(* Visualisation VISU_CFG_KEEL
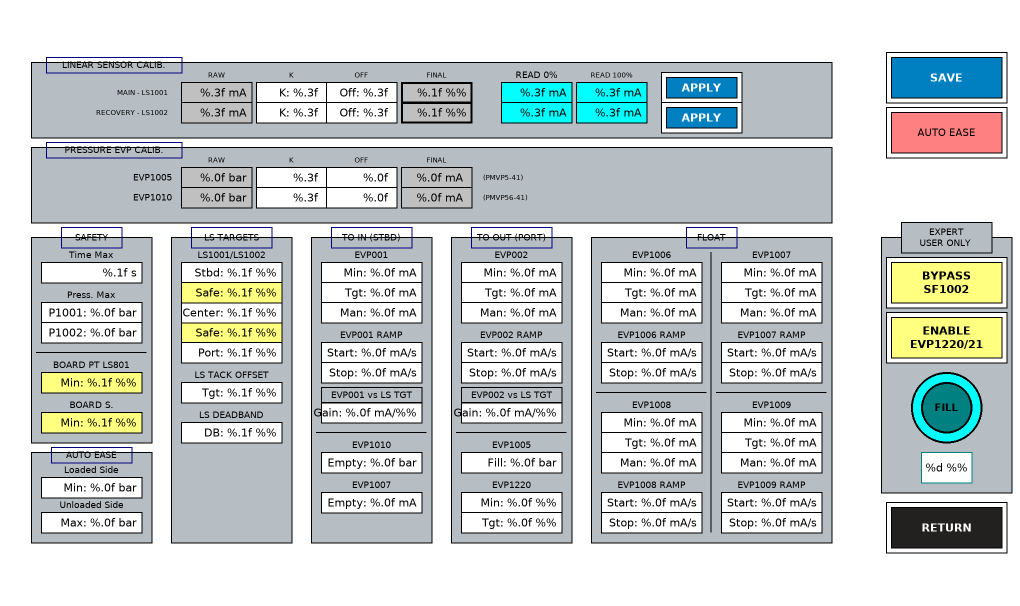
rectangle at (415,65)-(486,81): text "FINAL"
rectangle at (485,225)-(566,246): text "TO OUT (PORT)"
rectangle at (345,225)-(426,246): text "TO IN (STBD)"
rectangle at (20,550)-(331,601): text "%s"; shows INPUTS.sVisuTime
rounded rectangle at (905,55)-(1016,96): text "SAVE"; alarm colour if PARAMS.Save; toggles PARAMS.Save
rounded rectangle at (905,505)-(1016,546): text "RETURN"; opens VISU_2_KEEL
rectangle at (730,550)-(896,601): text "SAVED!"; invisible if PARAMS.Saved
rectangle at (20,0)-(426,51): text "CFG: KEEL"
rectangle at (55,260)-(156,281): text "%.1f s"; shows PARAMS.stKeelCfg.TimeMax; runs INTERN ASSIGN INPUTS.PresSelCalStbd[9]:=(FALSE); editable
rectangle at (65,245)-(146,261): text "Time Max"
rectangle at (55,300)-(156,321): text "P1001: %.0f bar"; shows P1001.MaxBar; runs INTERN ASSIGN INPUTS.PresSelCalStbd[9]:=(FALSE); editable
rectangle at (55,285)-(156,301): text "Press. Max"
rectangle at (55,320)-(156,341): text "P1002: %.0f bar"; shows P1002.MaxBar; runs INTERN ASSIGN INPUTS.PresSelCalStbd[9]:=(FALSE); editable
rectangle at (195,150)-(266,166): text "RAW"
rectangle at (415,150)-(486,166): text "FINAL"
rectangle at (270,150)-(341,166): text "K"
rectangle at (340,150)-(411,166): text "OFF"
rectangle at (415,165)-(486,186): text "%.0f mA"; shows EVP1005.mA; runs INTERN ASSIGN INPUTS.PresSelCalStbd[9]:=(FALSE)
rectangle at (270,165)-(341,186): text "%.3f"; shows EVP1005.Cal_K; runs INTERN ASSIGN INPUTS.PresSelCalStbd[9]:=(FALSE); editable
rectangle at (195,165)-(266,186): text "%.0f bar"; shows EVP1005.Bar; runs INTERN ASSIGN INPUTS.PresSelCalStbd[9]:=(FALSE)
rectangle at (340,165)-(411,186): text "%.0f"; shows EVP1005.Cal_Off; runs INTERN ASSIGN INPUTS.PresSelCalStbd[9]:=(FALSE); editable
rectangle at (145,165)-(196,186): text "EVP1005"
rectangle at (415,185)-(486,206): text "%.0f mA"; shows EVP1010.mA; runs INTERN ASSIGN INPUTS.PresSelCalStbd[9]:=(FALSE)
rectangle at (270,185)-(341,206): text "%.3f"; shows EVP1010.Cal_K; runs INTERN ASSIGN INPUTS.PresSelCalStbd[9]:=(FALSE); editable
rectangle at (195,185)-(266,206): text "%.0f bar"; shows EVP1010.Bar; runs INTERN ASSIGN INPUTS.PresSelCalStbd[9]:=(FALSE)
rectangle at (340,185)-(411,206): text "%.0f"; shows EVP1010.Cal_Off; runs INTERN ASSIGN INPUTS.PresSelCalStbd[9]:=(FALSE); editable
rectangle at (495,165)-(561,186): text "(PMVP5-41)"
rectangle at (145,185)-(196,206): text "EVP1010"
rectangle at (495,185)-(561,206): text "(PMVP56-41)"
ellipse at (925,370)-(996,441): alarm colour if MAIN.fbKeel.EVP_Fill = 0
ellipse at (935,380)-(986,431): text "FILL"; alarm colour if MAIN.fbKeel.IN_Hmi_fill; taps MAIN.fbKeel.IN_Hmi_fill
rounded rectangle at (905,315)-(1016,356): text "ENABLE / EVP1220/21"; alarm colour if MAIN.fbKEEL.EnableFill; toggles MAIN.fbKEEL.EnableFill
rounded rectangle at (915,220)-(1006,251): text "EXPERT / USER ONLY"
rounded rectangle at (680,75)-(751,96): text "APPLY"; toggles LS1001.Cal_Apply
rectangle at (590,80)-(661,101): text "%.3f mA"; shows LS1001.Cal_Max; alarm colour if LS1001.Cal_Max = 0.0; runs INTERN ASSIGN INPUTS.PresSelCalStbd[9]:=(FALSE); editable
rectangle at (515,80)-(586,101): text "%.3f mA"; shows LS1001.Cal_Min; alarm colour if LS1001.Cal_Min = 0.0; runs INTERN ASSIGN INPUTS.PresSelCalStbd[9]:=(FALSE); editable
rectangle at (55,80)-(186,101): text "MAIN - LS1001"
rectangle at (270,80)-(341,101): text "K: %.3f"; shows LS1001.Cal_K; runs INTERN ASSIGN INPUTS.PresSelCalStbd[9]:=(FALSE); editable
rectangle at (195,80)-(266,101): text "%.3f mA"; shows LS1001.Raw; alarm colour if LS1001.Err; runs INTERN ASSIGN INPUTS.PresSelCalStbd[9]:=(FALSE)
rectangle at (340,80)-(411,101): text "Off: %.3f"; shows LS1001.Cal_Off; runs INTERN ASSIGN INPUTS.PresSelCalStbd[9]:=(FALSE); editable
rectangle at (415,80)-(486,101): text "%.1f %%"; shows LS1001.Pos; runs INTERN ASSIGN INPUTS.PresSelCalStbd[9]:=(FALSE)
rectangle at (515,65)-(586,81): text "READ 0%"
rectangle at (590,65)-(661,81): text "READ 100%"
rounded rectangle at (680,105)-(751,126): text "APPLY"; toggles LS1002.Cal_Apply
rectangle at (590,100)-(661,121): text "%.3f mA"; shows LS1002.Cal_Max; alarm colour if LS1002.Cal_Max = 0.0; runs INTERN ASSIGN INPUTS.PresSelCalStbd[9]:=(FALSE); editable
rectangle at (515,100)-(586,121): text "%.3f mA"; shows LS1002.Cal_Min; alarm colour if LS1002.Cal_Min = 0.0; runs INTERN ASSIGN INPUTS.PresSelCalStbd[9]:=(FALSE); editable
rectangle at (55,100)-(186,121): text "RECOVERY - LS1002"
rectangle at (270,100)-(341,121): text "K: %.3f"; shows LS1002.Cal_K; runs INTERN ASSIGN INPUTS.PresSelCalStbd[9]:=(FALSE); editable
rectangle at (195,100)-(266,121): text "%.3f mA"; shows LS1002.Raw; alarm colour if LS1002.Err; runs INTERN ASSIGN INPUTS.PresSelCalStbd[9]:=(FALSE)
rectangle at (340,100)-(411,121): text "Off: %.3f"; shows LS1002.Cal_Off; runs INTERN ASSIGN INPUTS.PresSelCalStbd[9]:=(FALSE); editable
rectangle at (415,100)-(486,121): text "%.1f %%"; shows LS1002.Pos; runs INTERN ASSIGN INPUTS.PresSelCalStbd[9]:=(FALSE)
rounded rectangle at (905,260)-(1016,301): text "BYPASS / SF1002"; alarm colour if MAIN.fbKEEL.BypassSF; toggles MAIN.fbKEEL.BypassSF
rectangle at (55,370)-(156,391): text "Min: %.1f %%"; shows PARAMS.stKeelCfg.Board_P_Min_Out; runs INTERN ASSIGN INPUTS.PresSelCalStbd[9]:=(FALSE); editable
rectangle at (55,355)-(156,371): text "BOARD PT LS801"
rectangle at (55,410)-(156,431): text "Min: %.1f %%"; shows PARAMS.stKeelCfg.Board_S_Min_Out; runs INTERN ASSIGN INPUTS.PresSelCalStbd[9]:=(FALSE); editable
rectangle at (55,395)-(156,411): text "BOARD S."
rounded rectangle at (935,450)-(986,481): text "%d %%"; shows MAIN.fbKEEL.IN_Hmi_fill_Perc; editable 5..100
rectangle at (195,260)-(296,281): text "Stbd: %.1f %%"; shows PARAMS.stKeelCfg.TgtLS_In; runs INTERN ASSIGN INPUTS.PresSelCalStbd[9]:=(FALSE); editable
rectangle at (195,245)-(296,261): text "LS1001/LS1002"
rectangle at (195,320)-(296,341): text "Safe: %.1f %%"; shows PARAMS.stKeelCfg.TgtLS_Safe_Out; runs INTERN ASSIGN INPUTS.PresSelCalStbd[9]:=(FALSE); editable
rectangle at (195,300)-(296,321): text "Center: %.1f %%"; shows PARAMS.stKeelCfg.TgtLS_Mid; runs INTERN ASSIGN INPUTS.PresSelCalStbd[9]:=(FALSE); editable
rectangle at (195,280)-(296,301): text "Safe: %.1f %%"; shows PARAMS.stKeelCfg.TgtLS_Safe_In; runs INTERN ASSIGN INPUTS.PresSelCalStbd[9]:=(FALSE); editable
rectangle at (195,340)-(296,361): text "Port: %.1f %%"; shows PARAMS.stKeelCfg.TgtLS_Out; runs INTERN ASSIGN INPUTS.PresSelCalStbd[9]:=(FALSE); editable
rectangle at (195,420)-(296,441): text "DB: %.1f %%"; shows PARAMS.stKeelCfg.LS_DB; runs INTERN ASSIGN INPUTS.PresSelCalStbd[9]:=(FALSE); editable
rectangle at (195,405)-(296,421): text "LS DEADBAND"
rectangle at (615,260)-(716,281): text "Min: %.0f mA"; shows PARAMS.stKeelCfg.EVP_In_SE_Min; runs INTERN ASSIGN INPUTS.PresSelCalStbd[9]:=(FALSE); editable
rectangle at (615,245)-(716,261): text "EVP1006"
rectangle at (615,280)-(716,301): text "Tgt: %.0f mA"; shows PARAMS.stKeelCfg.EVP_In_SE_Max; runs INTERN ASSIGN INPUTS.PresSelCalStbd[9]:=(FALSE); editable
rectangle at (615,300)-(716,321): text "Man: %.0f mA"; shows PARAMS.stKeelCfg.EVP_In_SE_Man; runs INTERN ASSIGN INPUTS.PresSelCalStbd[9]:=(FALSE); editable
rectangle at (615,410)-(716,431): text "Min: %.0f mA"; shows PARAMS.stKeelCfg.EVP_In_FE_Min; runs INTERN ASSIGN INPUTS.PresSelCalStbd[9]:=(FALSE); editable
rectangle at (615,395)-(716,411): text "EVP1008"
rectangle at (615,430)-(716,451): text "Tgt: %.0f mA"; shows PARAMS.stKeelCfg.EVP_In_FE_Max; runs INTERN ASSIGN INPUTS.PresSelCalStbd[9]:=(FALSE); editable
rectangle at (615,450)-(716,471): text "Man: %.0f mA"; shows PARAMS.stKeelCfg.EVP_In_FE_Man; runs INTERN ASSIGN INPUTS.PresSelCalStbd[9]:=(FALSE); editable
rectangle at (335,260)-(436,281): text "Min: %.0f mA"; shows PARAMS.stKeelCfg.EVP_In_Eng_Min; runs INTERN ASSIGN INPUTS.PresSelCalStbd[9]:=(FALSE); editable
rectangle at (335,245)-(436,261): text "EVP001"
rectangle at (335,280)-(436,301): text "Tgt: %.0f mA"; shows PARAMS.stKeelCfg.EVP_In_Eng_Max; runs INTERN ASSIGN INPUTS.PresSelCalStbd[9]:=(FALSE); editable
rectangle at (335,300)-(436,321): text "Man: %.0f mA"; shows PARAMS.stKeelCfg.EVP_In_Eng_Man; runs INTERN ASSIGN INPUTS.PresSelCalStbd[9]:=(FALSE); editable
rectangle at (335,490)-(436,511): text "Empty: %.0f mA"; shows PARAMS.stKeelCfg.EVP_Out_SE_Empty; runs INTERN ASSIGN INPUTS.PresSelCalStbd[9]:=(FALSE); editable
rectangle at (335,475)-(436,491): text "EVP1007"
rectangle at (195,380)-(296,401): text "Tgt: %.1f %%"; shows PARAMS.stKeelCfg.TgtLS_Tack_Off; runs INTERN ASSIGN INPUTS.PresSelCalStbd[9]:=(FALSE); editable
rectangle at (195,365)-(296,381): text "LS TACK OFFSET"
rectangle at (335,450)-(436,471): text "Empty: %.0f bar"; shows PARAMS.stKeelCfg.EVP_In_P_Empty; runs INTERN ASSIGN INPUTS.PresSelCalStbd[9]:=(FALSE); editable
rectangle at (335,435)-(436,451): text "EVP1010"
rectangle at (475,260)-(576,281): text "Min: %.0f mA"; shows PARAMS.stKeelCfg.EVP_Out_Eng_Min; runs INTERN ASSIGN INPUTS.PresSelCalStbd[9]:=(FALSE); editable
rectangle at (475,245)-(576,261): text "EVP002"
rectangle at (475,280)-(576,301): text "Tgt: %.0f mA"; shows PARAMS.stKeelCfg.EVP_Out_Eng_Max; runs INTERN ASSIGN INPUTS.PresSelCalStbd[9]:=(FALSE); editable
rectangle at (475,300)-(576,321): text "Man: %.0f mA"; shows PARAMS.stKeelCfg.EVP_Out_Eng_Man; runs INTERN ASSIGN INPUTS.PresSelCalStbd[9]:=(FALSE); editable
rectangle at (475,450)-(576,471): text "Fill: %.0f bar"; shows PARAMS.stKeelCfg.EVP_Out_P_Fill; runs INTERN ASSIGN INPUTS.PresSelCalStbd[9]:=(FALSE); editable
rectangle at (475,435)-(576,451): text "EVP1005"
rectangle at (475,490)-(576,511): text "Min: %.0f %%"; shows PARAMS.stKeelCfg.EVP_Out_Fill_Min; runs INTERN ASSIGN INPUTS.PresSelCalStbd[9]:=(FALSE); editable
rectangle at (475,475)-(576,491): text "EVP1220"
rectangle at (475,510)-(576,531): text "Tgt: %.0f %%"; shows PARAMS.stKeelCfg.EVP_Out_Fill_Max; runs INTERN ASSIGN INPUTS.PresSelCalStbd[9]:=(FALSE); editable
rectangle at (735,260)-(836,281): text "Min: %.0f mA"; shows PARAMS.stKeelCfg.EVP_Out_SE_Min; runs INTERN ASSIGN INPUTS.PresSelCalStbd[9]:=(FALSE); editable
rectangle at (735,245)-(836,261): text "EVP1007"
rectangle at (735,280)-(836,301): text "Tgt: %.0f mA"; shows PARAMS.stKeelCfg.EVP_Out_SE_Max; runs INTERN ASSIGN INPUTS.PresSelCalStbd[9]:=(FALSE); editable
rectangle at (735,300)-(836,321): text "Man: %.0f mA"; shows PARAMS.stKeelCfg.EVP_Out_SE_Man; runs INTERN ASSIGN INPUTS.PresSelCalStbd[9]:=(FALSE); editable
rectangle at (735,410)-(836,431): text "Min: %.0f mA"; shows PARAMS.stKeelCfg.EVP_Out_FE_Min; runs INTERN ASSIGN INPUTS.PresSelCalStbd[9]:=(FALSE); editable
rectangle at (735,395)-(836,411): text "EVP1009"
rectangle at (735,430)-(836,451): text "Tgt: %.0f mA"; shows PARAMS.stKeelCfg.EVP_Out_FE_Max; runs INTERN ASSIGN INPUTS.PresSelCalStbd[9]:=(FALSE); editable
rectangle at (735,450)-(836,471): text "Man: %.0f mA"; shows PARAMS.stKeelCfg.EVP_Out_FE_Man; runs INTERN ASSIGN INPUTS.PresSelCalStbd[9]:=(FALSE); editable
rectangle at (335,340)-(436,361): text "Start: %.0f mA/s"; shows PARAMS.stKeelCfg.EVP_In_Eng_Inc; runs INTERN ASSIGN INPUTS.PresSelCalStbd[9]:=(FALSE); editable
rectangle at (335,325)-(436,341): text "EVP001 RAMP"
rectangle at (335,360)-(436,381): text "Stop: %.0f mA/s"; shows PARAMS.stKeelCfg.EVP_In_Eng_Dec; runs INTERN ASSIGN INPUTS.PresSelCalStbd[9]:=(FALSE); editable
rectangle at (475,340)-(576,361): text "Start: %.0f mA/s"; shows PARAMS.stKeelCfg.EVP_Out_Eng_Inc; runs INTERN ASSIGN INPUTS.PresSelCalStbd[9]:=(FALSE); editable
rectangle at (475,325)-(576,341): text "EVP002 RAMP"
rectangle at (475,360)-(576,381): text "Stop: %.0f mA/s"; shows PARAMS.stKeelCfg.EVP_Out_Eng_Dec; runs INTERN ASSIGN INPUTS.PresSelCalStbd[9]:=(FALSE); editable
rectangle at (615,340)-(716,361): text "Start: %.0f mA/s"; shows PARAMS.stKeelCfg.EVP_In_SE_Inc; runs INTERN ASSIGN INPUTS.PresSelCalStbd[9]:=(FALSE); editable
rectangle at (615,325)-(716,341): text "EVP1006 RAMP"
rectangle at (615,360)-(716,381): text "Stop: %.0f mA/s"; shows PARAMS.stKeelCfg.EVP_In_SE_Dec; runs INTERN ASSIGN INPUTS.PresSelCalStbd[9]:=(FALSE); editable
rectangle at (735,340)-(836,361): text "Start: %.0f mA/s"; shows PARAMS.stKeelCfg.EVP_Out_SE_Inc; runs INTERN ASSIGN INPUTS.PresSelCalStbd[9]:=(FALSE); editable
rectangle at (735,325)-(836,341): text "EVP1007 RAMP"
rectangle at (735,360)-(836,381): text "Stop: %.0f mA/s"; shows PARAMS.stKeelCfg.EVP_Out_SE_Dec; runs INTERN ASSIGN INPUTS.PresSelCalStbd[9]:=(FALSE); editable
rectangle at (615,490)-(716,511): text "Start: %.0f mA/s"; shows PARAMS.stKeelCfg.EVP_In_FE_Inc; runs INTERN ASSIGN INPUTS.PresSelCalStbd[9]:=(FALSE); editable
rectangle at (615,475)-(716,491): text "EVP1008 RAMP"
rectangle at (615,510)-(716,531): text "Stop: %.0f mA/s"; shows PARAMS.stKeelCfg.EVP_In_FE_Dec; runs INTERN ASSIGN INPUTS.PresSelCalStbd[9]:=(FALSE); editable
rectangle at (735,490)-(836,511): text "Start: %.0f mA/s"; shows PARAMS.stKeelCfg.EVP_Out_FE_Inc; runs INTERN ASSIGN INPUTS.PresSelCalStbd[9]:=(FALSE); editable
rectangle at (735,475)-(836,491): text "EVP1009 RAMP"
rectangle at (735,510)-(836,531): text "Stop: %.0f mA/s"; shows PARAMS.stKeelCfg.EVP_Out_FE_Dec; runs INTERN ASSIGN INPUTS.PresSelCalStbd[9]:=(FALSE); editable
rectangle at (335,400)-(436,421): text "Gain: %.0f mA/%%"; shows PARAMS.stKeelCfg.EVP_In_Eng_K; runs INTERN ASSIGN INPUTS.PresSelCalStbd[9]:=(FALSE); editable
rectangle at (335,385)-(436,401): text "EVP001 vs LS TGT"
rectangle at (475,400)-(576,421): text "Gain: %.0f mA/%%"; shows PARAMS.stKeelCfg.EVP_Out_Eng_K; runs INTERN ASSIGN INPUTS.PresSelCalStbd[9]:=(FALSE); editable
rectangle at (475,385)-(576,401): text "EVP002 vs LS TGT"
rectangle at (700,225)-(751,246): text "FLOAT"
rectangle at (195,65)-(266,81): text "RAW"
rectangle at (270,65)-(341,81): text "K"
rectangle at (340,65)-(411,81): text "OFF"
rectangle at (205,225)-(286,246): text "LS TARGETS"
rectangle at (75,225)-(136,246): text "SAFETY"
rectangle at (60,55)-(196,71): text "LINEAR SENSOR CALIB."
rectangle at (60,140)-(196,156): text "PRESSURE EVP CALIB."
rounded rectangle at (905,110)-(1016,151): text "AUTO EASE"; alarm colour if MAIN.aLP_Enable[20]; toggles MAIN.aLP_Enable[20]
rectangle at (65,445)-(146,461): text "AUTO EASE"
rectangle at (55,460)-(156,476): text "Loaded Side"
rectangle at (55,475)-(156,496): text "Min: %.0f bar"; shows PARAMS.stKeelCfg.MinLoadSide_Bar; runs INTERN ASSIGN INPUTS.PresSelCalStbd[9]:=(FALSE); editable
rectangle at (55,495)-(156,511): text "Unloaded Side"
rectangle at (55,510)-(156,531): text "Max: %.0f bar"; shows PARAMS.stKeelCfg.MaxUnloadSide_Bar; runs INTERN ASSIGN INPUTS.PresSelCalStbd[9]:=(FALSE); editable
22 more shapes without text or variables
*)

(* Visualisation VISU_CFG_POWERPACK
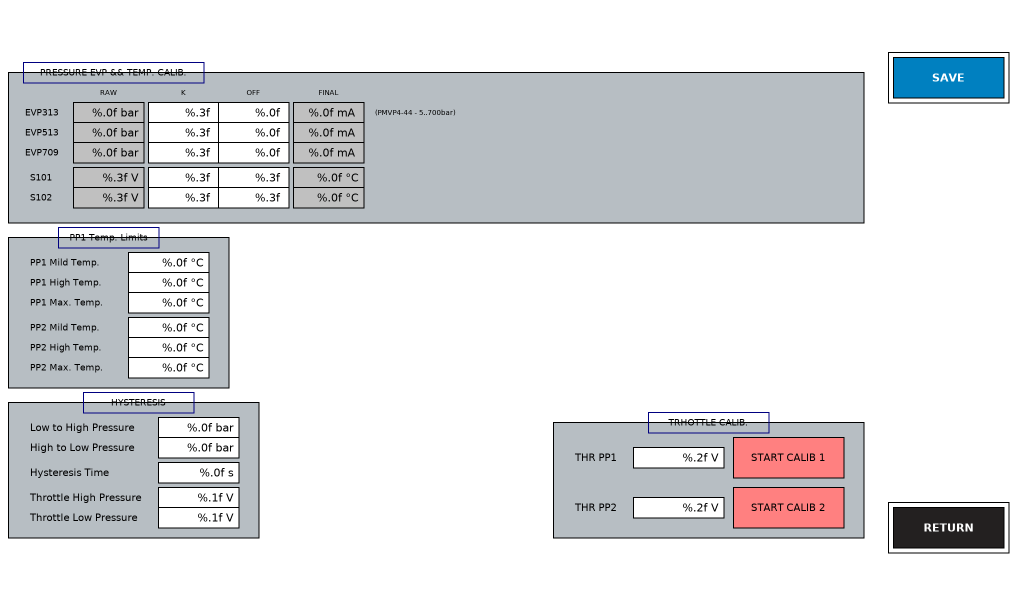
rectangle at (20,0)-(436,51): text "CFG: POWERPACK"
rectangle at (20,550)-(331,601): text "%s"; shows INPUTS.sVisuTime
rounded rectangle at (905,55)-(1016,96): text "SAVE"; alarm colour if PARAMS.Save; toggles PARAMS.Save
rounded rectangle at (905,505)-(1016,546): text "RETURN"; opens VISU_1_PUMPS
rectangle at (95,390)-(206,411): text "HYSTERESIS"
rectangle at (170,415)-(251,436): text "%.0f bar"; shows PARAMS.stPowerpackCfg.Hyst_HP; runs INTERN ASSIGN INPUTS.PresSelCalStbd[9]:=(FALSE); editable
rectangle at (170,435)-(251,456): text "%.0f bar"; shows PARAMS.stPowerpackCfg.Hyst_LP; runs INTERN ASSIGN INPUTS.PresSelCalStbd[9]:=(FALSE); editable
rectangle at (170,460)-(251,481): text "%.0f s"; shows PARAMS.stPowerpackCfg.Hyst_TM; runs INTERN ASSIGN INPUTS.PresSelCalStbd[9]:=(FALSE); editable
rectangle at (40,415)-(171,436): text "Low to High Pressure"; shows RECV_J1939.F004.DriverDemandTorque
rectangle at (40,435)-(171,456): text "High to Low Pressure"; shows RECV_J1939.F004.DriverDemandTorque
rectangle at (40,460)-(171,481): text "Hysteresis Time"; shows RECV_J1939.F004.DriverDemandTorque
rectangle at (730,550)-(896,601): text "SAVED!"; invisible if PARAMS.Saved
rectangle at (660,410)-(781,431): text "TRHOTTLE CALIB."
rounded rectangle at (745,435)-(856,476): text "START CALIB 1"; alarm colour if POWERPACK.Calib1; toggles POWERPACK.Calib1
rectangle at (645,445)-(736,466): text "%.2f V"; shows THR_PP1; runs INTERN ASSIGN INPUTS.PresSelCalStbd[9]:=(FALSE); editable
rectangle at (585,445)-(641,466): text "THR PP1"; shows RECV_J1939.F004.DriverDemandTorque
rectangle at (645,495)-(736,516): text "%.2f V"; shows THR_PP2; runs INTERN ASSIGN INPUTS.PresSelCalStbd[9]:=(FALSE); editable
rectangle at (585,495)-(641,516): text "THR PP2"; shows RECV_J1939.F004.DriverDemandTorque
rounded rectangle at (745,485)-(856,526): text "START CALIB 2"; alarm colour if POWERPACK.Calib2; toggles POWERPACK.Calib2
rectangle at (170,485)-(251,506): text "%.1f V"; shows PARAMS.stPowerpackCfg.Thr_HP; runs INTERN ASSIGN INPUTS.PresSelCalStbd[9]:=(FALSE); editable 1..5
rectangle at (40,485)-(171,506): text "Throttle High Pressure"; shows RECV_J1939.F004.DriverDemandTorque
rectangle at (170,505)-(251,526): text "%.1f V"; shows PARAMS.stPowerpackCfg.Thr_LP; runs INTERN ASSIGN INPUTS.PresSelCalStbd[9]:=(FALSE); editable 1..5
rectangle at (40,505)-(171,526): text "Throttle Low Pressure"; shows RECV_J1939.F004.DriverDemandTorque
rectangle at (85,80)-(156,101): text "RAW"
rectangle at (305,80)-(376,101): text "FINAL"
rectangle at (160,80)-(231,101): text "K"
rectangle at (230,80)-(301,101): text "OFF"
rectangle at (305,100)-(376,121): text "%.0f mA"; shows EVP313.mA; runs INTERN ASSIGN INPUTS.PresSelCalStbd[9]:=(FALSE)
rectangle at (160,100)-(231,121): text "%.3f"; shows EVP313.Cal_K; runs INTERN ASSIGN INPUTS.PresSelCalStbd[9]:=(FALSE); editable
rectangle at (85,100)-(156,121): text "%.0f bar"; shows EVP313.Bar; runs INTERN ASSIGN INPUTS.PresSelCalStbd[9]:=(FALSE)
rectangle at (230,100)-(301,121): text "%.0f"; shows EVP313.Cal_Off; runs INTERN ASSIGN INPUTS.PresSelCalStbd[9]:=(FALSE); editable
rectangle at (35,100)-(86,121): text "EVP313"
rectangle at (305,120)-(376,141): text "%.0f mA"; shows EVP513.mA; runs INTERN ASSIGN INPUTS.PresSelCalStbd[9]:=(FALSE)
rectangle at (160,120)-(231,141): text "%.3f"; shows EVP513.Cal_K; runs INTERN ASSIGN INPUTS.PresSelCalStbd[9]:=(FALSE); editable
rectangle at (85,120)-(156,141): text "%.0f bar"; shows EVP513.Bar; runs INTERN ASSIGN INPUTS.PresSelCalStbd[9]:=(FALSE)
rectangle at (230,120)-(301,141): text "%.0f"; shows EVP513.Cal_Off; runs INTERN ASSIGN INPUTS.PresSelCalStbd[9]:=(FALSE); editable
rectangle at (385,100)-(581,121): text "(PMVP4-44 - 5..700bar)"
rectangle at (305,140)-(376,161): text "%.0f mA"; shows EVP709.mA; runs INTERN ASSIGN INPUTS.PresSelCalStbd[9]:=(FALSE)
rectangle at (160,140)-(231,161): text "%.3f"; shows EVP709.Cal_K; runs INTERN ASSIGN INPUTS.PresSelCalStbd[9]:=(FALSE); editable
rectangle at (85,140)-(156,161): text "%.0f bar"; shows EVP709.Bar; runs INTERN ASSIGN INPUTS.PresSelCalStbd[9]:=(FALSE)
rectangle at (230,140)-(301,161): text "%.0f"; shows EVP709.Cal_Off; runs INTERN ASSIGN INPUTS.PresSelCalStbd[9]:=(FALSE); editable
rectangle at (35,120)-(86,141): text "EVP513"
rectangle at (35,140)-(86,161): text "EVP709"
rectangle at (35,60)-(216,81): text "PRESSURE EVP && TEMP. CALIB."
rectangle at (40,250)-(121,271): text "PP1 Mild Temp."
rectangle at (140,250)-(221,271): text "%.0f °C"; shows S101.LowDeg; runs INTERN ASSIGN INPUTS.PresSelCalStbd[9]:=(FALSE); editable
rectangle at (40,270)-(121,291): text "PP1 High Temp."
rectangle at (140,270)-(221,291): text "%.0f °C"; shows S101.HigDeg; runs INTERN ASSIGN INPUTS.PresSelCalStbd[9]:=(FALSE); editable
rectangle at (70,225)-(171,246): text "PP1 Temp. Limits"
rectangle at (40,290)-(121,311): text "PP1 Max. Temp."
rectangle at (140,290)-(221,311): text "%.0f °C"; shows S101.MaxDeg; runs INTERN ASSIGN INPUTS.PresSelCalStbd[9]:=(FALSE); editable
rectangle at (40,165)-(86,186): text "S101"
rectangle at (305,165)-(376,186): text "%.0f °C"; shows S101.Deg
rectangle at (160,165)-(231,186): text "%.3f"; shows S101.Cal_K; runs INTERN ASSIGN INPUTS.PresSelCalStbd[9]:=(FALSE); editable
rectangle at (85,165)-(156,186): text "%.3f V"; shows S101.Raw; alarm colour if S101.Err; runs INTERN ASSIGN INPUTS.PresSelCalStbd[9]:=(FALSE)
rectangle at (230,165)-(301,186): text "%.3f"; shows S101.Cal_Off; runs INTERN ASSIGN INPUTS.PresSelCalStbd[9]:=(FALSE); editable
rectangle at (40,185)-(86,206): text "S102"
rectangle at (305,185)-(376,206): text "%.0f °C"; shows S102.Deg
rectangle at (160,185)-(231,206): text "%.3f"; shows S102.Cal_K; runs INTERN ASSIGN INPUTS.PresSelCalStbd[9]:=(FALSE); editable
rectangle at (85,185)-(156,206): text "%.3f V"; shows S102.Raw; alarm colour if S102.Err; runs INTERN ASSIGN INPUTS.PresSelCalStbd[9]:=(FALSE)
rectangle at (230,185)-(301,206): text "%.3f"; shows S102.Cal_Off; runs INTERN ASSIGN INPUTS.PresSelCalStbd[9]:=(FALSE); editable
rectangle at (40,315)-(121,336): text "PP2 Mild Temp."
rectangle at (140,315)-(221,336): text "%.0f °C"; shows S102.LowDeg; runs INTERN ASSIGN INPUTS.PresSelCalStbd[9]:=(FALSE); editable
rectangle at (40,335)-(121,356): text "PP2 High Temp."
rectangle at (140,335)-(221,356): text "%.0f °C"; shows S102.HigDeg; runs INTERN ASSIGN INPUTS.PresSelCalStbd[9]:=(FALSE); editable
rectangle at (40,355)-(121,376): text "PP2 Max. Temp."
rectangle at (140,355)-(221,376): text "%.0f °C"; shows S102.MaxDeg; runs INTERN ASSIGN INPUTS.PresSelCalStbd[9]:=(FALSE); editable
6 more shapes without text or variables
*)

(* Visualisation VISU_CFG_PROPULSION
rectangle at (55,305)-(116,326): text "PROP"
rounded rectangle at (905,505)-(1016,546): text "RETURN"; opens VISU_1_ENGINE
rectangle at (20,0)-(331,51): text "CFG: PROPULSION"
rectangle at (305,185)-(376,206): text "%.0f rpm"; shows PARAMS.stPropulsionCfg.aEng_RPM[10]; editable
rectangle at (380,185)-(451,206): text "%.0f mA"; shows PARAMS.stPropulsionCfg.aEVP_mA[10]; editable
rectangle at (195,185)-(226,206): text "100%"
rectangle at (230,185)-(301,206): text "%.2f V"; shows PARAMS.stPropulsionCfg.aThrt_V[10]; runs INTERN ASSIGN INPUTS.PresSelCalStbd[9]:=(FALSE); editable
rectangle at (230,365)-(301,386): text "%.2f V"; shows PARAMS.stPropulsionCfg.aThrt_V[0]; runs INTERN ASSIGN INPUTS.PresSelCalStbd[9]:=(FALSE); editable
rectangle at (195,105)-(226,126): text "0%"
rectangle at (230,105)-(301,126): text "%.2f V"; shows PARAMS.stPropulsionCfg.aThrt_V[6]; editable
rectangle at (230,285)-(301,306): text "%.2f V"; shows PARAMS.stPropulsionCfg.aThrt_V[4]; runs INTERN ASSIGN INPUTS.PresSelCalStbd[9]:=(FALSE); editable
rectangle at (195,165)-(226,186): text "75%"
rectangle at (195,145)-(226,166): text "50%"
rectangle at (195,125)-(226,146): text "25%"
rectangle at (230,85)-(301,106): text "THROTTLE"
rectangle at (305,85)-(376,106): text "ENGINE"
rectangle at (380,85)-(451,106): text "PROPELLER"
rectangle at (305,165)-(376,186): text "%.0f rpm"; shows PARAMS.stPropulsionCfg.aEng_RPM[9]; editable
rectangle at (305,145)-(376,166): text "%.0f rpm"; shows PARAMS.stPropulsionCfg.aEng_RPM[8]; editable
rectangle at (305,125)-(376,146): text "%.0f rpm"; shows PARAMS.stPropulsionCfg.aEng_RPM[7]; editable
rectangle at (305,105)-(376,126): text "%.0f rpm"; shows PARAMS.stPropulsionCfg.aEng_RPM[6]; editable
rectangle at (305,285)-(376,306): text "%.0f rpm"; shows PARAMS.stPropulsionCfg.aEng_RPM[4]; editable
rectangle at (305,305)-(376,326): text "%.0f rpm"; shows PARAMS.stPropulsionCfg.aEng_RPM[3]; editable
rectangle at (305,325)-(376,346): text "%.0f rpm"; shows PARAMS.stPropulsionCfg.aEng_RPM[2]; editable
rectangle at (305,345)-(376,366): text "%.0f rpm"; shows PARAMS.stPropulsionCfg.aEng_RPM[1]; editable
rectangle at (305,365)-(376,386): text "%.0f rpm"; shows PARAMS.stPropulsionCfg.aEng_RPM[0]; editable
rectangle at (230,125)-(301,146): text "%.2f V"; shows PARAMS.stPropulsionCfg.aThrt_V[7]
rectangle at (230,145)-(301,166): text "%.2f V"; shows PARAMS.stPropulsionCfg.aThrt_V[8]
rectangle at (230,165)-(301,186): text "%.2f V"; shows PARAMS.stPropulsionCfg.aThrt_V[9]
rectangle at (230,305)-(301,326): text "%.2f V"; shows PARAMS.stPropulsionCfg.aThrt_V[3]
rectangle at (230,325)-(301,346): text "%.2f V"; shows PARAMS.stPropulsionCfg.aThrt_V[2]
rectangle at (230,345)-(301,366): text "%.2f V"; shows PARAMS.stPropulsionCfg.aThrt_V[1]
rectangle at (380,165)-(451,186): text "%.0f mA"; shows PARAMS.stPropulsionCfg.aEVP_mA[9]; editable
rectangle at (380,145)-(451,166): text "%.0f mA"; shows PARAMS.stPropulsionCfg.aEVP_mA[8]; editable
rectangle at (380,125)-(451,146): text "%.0f mA"; shows PARAMS.stPropulsionCfg.aEVP_mA[7]; editable
rectangle at (380,105)-(451,126): text "%.0f mA"; shows PARAMS.stPropulsionCfg.aEVP_mA[6]; editable
rectangle at (380,285)-(451,306): text "%.0f mA"; shows PARAMS.stPropulsionCfg.aEVP_mA[4]; editable
rectangle at (290,240)-(391,261): text "REVERSE"
rectangle at (380,305)-(451,326): text "%.0f mA"; shows PARAMS.stPropulsionCfg.aEVP_mA[3]; editable
rectangle at (380,325)-(451,346): text "%.0f mA"; shows PARAMS.stPropulsionCfg.aEVP_mA[2]; editable
rectangle at (380,345)-(451,366): text "%.0f mA"; shows PARAMS.stPropulsionCfg.aEVP_mA[1]; editable
rectangle at (380,365)-(451,386): text "%.0f mA"; shows PARAMS.stPropulsionCfg.aEVP_mA[0]; editable
rectangle at (0,0)-(1,1): text "{ExtendedElement},Visu\ElementDLL.ete,1,@Bargraph,76,131,1,1,0,PARAMS.stPropulsionCfg.aEng_RPM[10],,%,200,400,800,2400,0,0,0,0,0,0,0,-13,16,700,Arial,0,255,0,255,0,0,0,0,0,0,0,0,0,,0,"
rectangle at (12,65)-(28,122): alarm colour if (PARAMS.stPropulsionCfg.aEng_RPM[10]) < 0; top ((PARAMS.stPropulsionCfg.aEng_RPM[10] * 1.0) - 1600)  * -0.07125
rectangle at (0,0)-(1,1): text "{ExtendedElement},Visu\ElementDLL.ete,1,@Bargraph,76,131,1,1,0,PARAMS.stPropulsionCfg.aEng_RPM[9],,%,200,400,800,2400,0,0,0,0,0,0,0,-13,16,700,Arial,0,255,0,255,0,0,0,0,0,0,0,0,0,,0,"
rectangle at (12,65)-(28,122): alarm colour if (PARAMS.stPropulsionCfg.aEng_RPM[9]) < 0; top ((PARAMS.stPropulsionCfg.aEng_RPM[9] * 1.0) - 1600)  * -0.07125
rectangle at (0,0)-(1,1): text "{ExtendedElement},Visu\ElementDLL.ete,1,@Bargraph,76,131,1,1,0,PARAMS.stPropulsionCfg.aEng_RPM[8],,%,200,400,800,2400,0,0,0,0,0,0,0,-13,16,700,Arial,0,255,0,255,0,0,0,0,0,0,0,0,0,,0,"
rectangle at (12,65)-(28,122): alarm colour if (PARAMS.stPropulsionCfg.aEng_RPM[8]) < 0; top ((PARAMS.stPropulsionCfg.aEng_RPM[8] * 1.0) - 1600)  * -0.07125
rectangle at (0,0)-(1,1): text "{ExtendedElement},Visu\ElementDLL.ete,1,@Bargraph,76,131,1,1,0,PARAMS.stPropulsionCfg.aEng_RPM[7],,%,200,400,800,2400,0,0,0,0,0,0,0,-13,16,700,Arial,0,255,0,255,0,0,0,0,0,0,0,0,0,,0,"
rectangle at (12,65)-(28,122): alarm colour if (PARAMS.stPropulsionCfg.aEng_RPM[7]) < 0; top ((PARAMS.stPropulsionCfg.aEng_RPM[7] * 1.0) - 1600)  * -0.07125
rectangle at (0,0)-(1,1): text "{ExtendedElement},Visu\ElementDLL.ete,1,@Bargraph,76,131,1,1,0,PARAMS.stPropulsionCfg.aEng_RPM[6],,%,200,400,800,2400,0,0,0,0,0,0,0,-13,16,700,Arial,0,255,0,255,0,0,0,0,0,0,0,0,0,,0,"
rectangle at (12,65)-(28,122): alarm colour if (PARAMS.stPropulsionCfg.aEng_RPM[6]) < 0; top ((PARAMS.stPropulsionCfg.aEng_RPM[6] * 1.0) - 1600)  * -0.07125
rectangle at (455,80)-(486,101): text "2400"
rectangle at (455,110)-(486,131): text "2000"
rectangle at (455,140)-(486,161): text "1600"
rectangle at (455,170)-(486,191): text "1200"
rectangle at (455,200)-(486,221): text "800"
rectangle at (0,0)-(1,1): text "{ExtendedElement},Visu\ElementDLL.ete,1,@Bargraph,76,131,1,1,0,PARAMS.stPropulsionCfg.aEng_RPM[0],,%,200,400,800,2400,0,0,0,0,0,0,0,-13,16,700,Arial,0,255,0,255,0,0,0,0,0,0,0,0,0,,0,"
rectangle at (12,65)-(28,122): alarm colour if (PARAMS.stPropulsionCfg.aEng_RPM[0]) < 0; top ((PARAMS.stPropulsionCfg.aEng_RPM[0] * 1.0) - 1600)  * -0.07125
rectangle at (0,0)-(1,1): text "{ExtendedElement},Visu\ElementDLL.ete,1,@Bargraph,76,131,1,1,0,PARAMS.stPropulsionCfg.aEng_RPM[1],,%,200,400,800,2400,0,0,0,0,0,0,0,-13,16,700,Arial,0,255,0,255,0,0,0,0,0,0,0,0,0,,0,"
rectangle at (12,65)-(28,122): alarm colour if (PARAMS.stPropulsionCfg.aEng_RPM[1]) < 0; top ((PARAMS.stPropulsionCfg.aEng_RPM[1] * 1.0) - 1600)  * -0.07125
rectangle at (0,0)-(1,1): text "{ExtendedElement},Visu\ElementDLL.ete,1,@Bargraph,76,131,1,1,0,PARAMS.stPropulsionCfg.aEng_RPM[2],,%,200,400,800,2400,0,0,0,0,0,0,0,-13,16,700,Arial,0,255,0,255,0,0,0,0,0,0,0,0,0,,0,"
rectangle at (12,65)-(28,122): alarm colour if (PARAMS.stPropulsionCfg.aEng_RPM[2]) < 0; top ((PARAMS.stPropulsionCfg.aEng_RPM[2] * 1.0) - 1600)  * -0.07125
rectangle at (0,0)-(1,1): text "{ExtendedElement},Visu\ElementDLL.ete,1,@Bargraph,76,131,1,1,0,PARAMS.stPropulsionCfg.aEng_RPM[3],,%,200,400,800,2400,0,0,0,0,0,0,0,-13,16,700,Arial,0,255,0,255,0,0,0,0,0,0,0,0,0,,0,"
rectangle at (12,65)-(28,122): alarm colour if (PARAMS.stPropulsionCfg.aEng_RPM[3]) < 0; top ((PARAMS.stPropulsionCfg.aEng_RPM[3] * 1.0) - 1600)  * -0.07125
rectangle at (0,0)-(1,1): text "{ExtendedElement},Visu\ElementDLL.ete,1,@Bargraph,76,131,1,1,0,PARAMS.stPropulsionCfg.aEng_RPM[4],,%,200,400,800,2400,0,0,0,0,0,0,0,-13,16,700,Arial,0,255,0,255,0,0,0,0,0,0,0,0,0,,0,"
rectangle at (12,65)-(28,122): alarm colour if (PARAMS.stPropulsionCfg.aEng_RPM[4]) < 0; top ((PARAMS.stPropulsionCfg.aEng_RPM[4] * 1.0) - 1600)  * -0.07125
rectangle at (490,60)-(561,81): text "ENG. RPM"
rectangle at (490,240)-(561,261): text "ENG. RPM"
rectangle at (0,0)-(1,1): text "{ExtendedElement},Visu\ElementDLL.ete,1,@Bargraph,76,131,1,1,0,PARAMS.stPropulsionCfg.aEVP_mA[6],,%,62.5,125,200,700,0,0,0,0,0,0,0,-13,16,700,Arial,255,0,0,255,0,0,0,0,0,0,0,0,0,,0,"
rectangle at (12,65)-(28,122): alarm colour if (PARAMS.stPropulsionCfg.aEVP_mA[6]) < 0; top ((PARAMS.stPropulsionCfg.aEVP_mA[6] * 1.0) - 450)  * -0.228
rectangle at (600,60)-(671,81): text "PROP. mA"
rectangle at (565,80)-(596,101): text "700"
rectangle at (565,110)-(596,131): text "575"
rectangle at (565,140)-(596,161): text "450"
rectangle at (565,170)-(596,191): text "325"
rectangle at (565,200)-(596,221): text "200"
rectangle at (0,0)-(1,1): text "{ExtendedElement},Visu\ElementDLL.ete,1,@Bargraph,76,131,1,1,0,PARAMS.stPropulsionCfg.aEVP_mA[7],,%,62.5,125,200,700,0,0,0,0,0,0,0,-13,16,700,Arial,255,0,0,255,0,0,0,0,0,0,0,0,0,,0,"
rectangle at (12,65)-(28,122): alarm colour if (PARAMS.stPropulsionCfg.aEVP_mA[7]) < 0; top ((PARAMS.stPropulsionCfg.aEVP_mA[7] * 1.0) - 450)  * -0.228
rectangle at (0,0)-(1,1): text "{ExtendedElement},Visu\ElementDLL.ete,1,@Bargraph,76,131,1,1,0,PARAMS.stPropulsionCfg.aEVP_mA[8],,%,62.5,125,200,700,0,0,0,0,0,0,0,-13,16,700,Arial,255,0,0,255,0,0,0,0,0,0,0,0,0,,0,"
rectangle at (12,65)-(28,122): alarm colour if (PARAMS.stPropulsionCfg.aEVP_mA[8]) < 0; top ((PARAMS.stPropulsionCfg.aEVP_mA[8] * 1.0) - 450)  * -0.228
rectangle at (0,0)-(1,1): text "{ExtendedElement},Visu\ElementDLL.ete,1,@Bargraph,76,131,1,1,0,PARAMS.stPropulsionCfg.aEVP_mA[9],,%,62.5,125,200,700,0,0,0,0,0,0,0,-13,16,700,Arial,255,0,0,255,0,0,0,0,0,0,0,0,0,,0,"
rectangle at (12,65)-(28,122): alarm colour if (PARAMS.stPropulsionCfg.aEVP_mA[9]) < 0; top ((PARAMS.stPropulsionCfg.aEVP_mA[9] * 1.0) - 450)  * -0.228
rectangle at (0,0)-(1,1): text "{ExtendedElement},Visu\ElementDLL.ete,1,@Bargraph,76,131,1,1,0,PARAMS.stPropulsionCfg.aEVP_mA[10],,%,62.5,125,200,700,0,0,0,0,0,0,0,-13,16,700,Arial,255,0,0,255,0,0,0,0,0,0,0,0,0,,0,"
rectangle at (12,65)-(28,122): alarm colour if (PARAMS.stPropulsionCfg.aEVP_mA[10]) < 0; top ((PARAMS.stPropulsionCfg.aEVP_mA[10] * 1.0) - 450)  * -0.228
rectangle at (0,0)-(1,1): text "{ExtendedElement},Visu\ElementDLL.ete,1,@Bargraph,76,131,1,1,0,PARAMS.stPropulsionCfg.aEVP_mA[4],,%,62.5,125,200,700,0,0,0,0,0,0,0,-13,16,700,Arial,255,0,0,255,0,0,0,0,0,0,0,0,0,,0,"
rectangle at (12,65)-(28,122): alarm colour if (PARAMS.stPropulsionCfg.aEVP_mA[4]) < 0; top ((PARAMS.stPropulsionCfg.aEVP_mA[4] * 1.0) - 450)  * -0.228
rectangle at (0,0)-(1,1): text "{ExtendedElement},Visu\ElementDLL.ete,1,@Bargraph,76,131,1,1,0,PARAMS.stPropulsionCfg.aEVP_mA[3],,%,62.5,125,200,700,0,0,0,0,0,0,0,-13,16,700,Arial,255,0,0,255,0,0,0,0,0,0,0,0,0,,0,"
rectangle at (12,65)-(28,122): alarm colour if (PARAMS.stPropulsionCfg.aEVP_mA[3]) < 0; top ((PARAMS.stPropulsionCfg.aEVP_mA[3] * 1.0) - 450)  * -0.228
rectangle at (0,0)-(1,1): text "{ExtendedElement},Visu\ElementDLL.ete,1,@Bargraph,76,131,1,1,0,PARAMS.stPropulsionCfg.aEVP_mA[2],,%,62.5,125,200,700,0,0,0,0,0,0,0,-13,16,700,Arial,255,0,0,255,0,0,0,0,0,0,0,0,0,,0,"
rectangle at (12,65)-(28,122): alarm colour if (PARAMS.stPropulsionCfg.aEVP_mA[2]) < 0; top ((PARAMS.stPropulsionCfg.aEVP_mA[2] * 1.0) - 450)  * -0.228
rectangle at (0,0)-(1,1): text "{ExtendedElement},Visu\ElementDLL.ete,1,@Bargraph,76,131,1,1,0,PARAMS.stPropulsionCfg.aEVP_mA[1],,%,62.5,125,200,700,0,0,0,0,0,0,0,-13,16,700,Arial,255,0,0,255,0,0,0,0,0,0,0,0,0,,0,"
rectangle at (12,65)-(28,122): alarm colour if (PARAMS.stPropulsionCfg.aEVP_mA[1]) < 0; top ((PARAMS.stPropulsionCfg.aEVP_mA[1] * 1.0) - 450)  * -0.228
rectangle at (0,0)-(1,1): text "{ExtendedElement},Visu\ElementDLL.ete,1,@Bargraph,76,131,1,1,0,PARAMS.stPropulsionCfg.aEVP_mA[0],,%,62.5,125,200,700,0,0,0,0,0,0,0,-13,16,700,Arial,255,0,0,255,0,0,0,0,0,0,0,0,0,,0,"
rectangle at (12,65)-(28,122): alarm colour if (PARAMS.stPropulsionCfg.aEVP_mA[0]) < 0; top ((PARAMS.stPropulsionCfg.aEVP_mA[0] * 1.0) - 450)  * -0.228
rectangle at (600,240)-(671,261): text "PROP. mA"
rectangle at (290,60)-(391,81): text "FORWARD"
rectangle at (230,265)-(301,286): text "THROTTLE"
rectangle at (305,265)-(376,286): text "ENGINE"
rectangle at (380,265)-(451,286): text "PROPELLER"
rectangle at (20,550)-(221,601): text "%s"; shows INPUTS.sVisuTime
rounded rectangle at (905,55)-(1016,96): text "SAVE"; alarm colour if PARAMS.Save; toggles PARAMS.Save
rectangle at (30,85)-(141,106): text "THR: %.2f V"; shows PARAMS.stPropulsionCfg.aThrt_V[5]; runs INTERN ASSIGN INPUTS.PresSelCalStbd[9]:=(FALSE); editable
rectangle at (30,350)-(141,371): text "PROP teeth: %.0f"; shows PARAMS.stPropulsionCfg.PropRPM_K; runs INTERN ASSIGN INPUTS.PresSelCalStbd[9]:=(FALSE); editable
rectangle at (30,165)-(141,186): text "THR: %.2f V"; shows ENGINE.fbPropulsion.Throttle_V; alarm colour if ENGINE.fbPropulsion.Throttle_err; runs INTERN ASSIGN INPUTS.PresSelCalStbd[9]:=(FALSE)
rectangle at (30,105)-(141,126): text "DB: %.2f V"; shows PARAMS.stPropulsionCfg.IdleDB_V; runs INTERN ASSIGN INPUTS.PresSelCalStbd[9]:=(FALSE); editable
rectangle at (60,60)-(111,81): text "IDLE"
rectangle at (30,185)-(141,206): text "THR: %.0f rpm"; shows ENGINE.fbPropulsion.Tgt_RPM; runs INTERN ASSIGN INPUTS.PresSelCalStbd[9]:=(FALSE)
rectangle at (30,330)-(141,351): text "PROP: %.0f rpm"; shows .Prop_RPM; runs INTERN ASSIGN INPUTS.PresSelCalStbd[9]:=(FALSE)
rectangle at (30,250)-(141,271): text "ENG: %.0f rpm"; shows RECV_J1939.F004.EngineActualSpeed; runs INTERN ASSIGN INPUTS.PresSelCalStbd[9]:=(FALSE)
rectangle at (30,270)-(141,291): text "ENG: %d %%"; shows RECV_J1939.F004.EngineActualTorque; runs INTERN ASSIGN INPUTS.PresSelCalStbd[9]:=(FALSE)
rectangle at (30,225)-(141,246): text "REV: %.d mA"; shows ENGINE.fbPropulsion.RevEVP; runs INTERN ASSIGN INPUTS.PresSelCalStbd[9]:=(FALSE)
rectangle at (30,205)-(141,226): text "FWD: %.d mA"; shows ENGINE.fbPropulsion.FwdEVP; runs INTERN ASSIGN INPUTS.PresSelCalStbd[9]:=(FALSE)
rounded rectangle at (905,220)-(1016,261): text "ENGINE / STOP"; alarm colour if ENGINE.Engine_STOP; taps ENGINE.Engine_STOP
rectangle at (730,550)-(896,601): text "SAVED!"; invisible if PARAMS.Saved
rectangle at (30,465)-(141,486): text "EV DLY: %.0f sec"; shows PARAMS.stPropulsionCfg.Delay_Off; runs INTERN ASSIGN INPUTS.PresSelCalStbd[9]:=(FALSE); editable 1..10
rectangle at (30,395)-(141,416): text "MAX: %.0f bar"; shows P1101.MaxBar; runs INTERN ASSIGN INPUTS.PresSelCalStbd[9]:=(FALSE); editable
rectangle at (30,440)-(141,461): text "MAX: %.0f bar"; shows P1102.MaxBar; runs INTERN ASSIGN INPUTS.PresSelCalStbd[9]:=(FALSE); editable
rectangle at (30,375)-(141,396): text "FWD: %.1f bar"; shows P1101.Bar; alarm colour if P1101.Alarm.Adver; runs INTERN ASSIGN INPUTS.PresSelCalStbd[9]:=(FALSE)
rectangle at (30,420)-(141,441): text "REV: %.1f bar"; shows P1102.Bar; alarm colour if P1102.Alarm.Adver; runs INTERN ASSIGN INPUTS.PresSelCalStbd[9]:=(FALSE)
rectangle at (195,365)-(226,386): text "100%"
rectangle at (195,285)-(226,306): text "0%"
rectangle at (195,345)-(226,366): text "75%"
rectangle at (195,325)-(226,346): text "50%"
rectangle at (195,305)-(226,326): text "25%"
rectangle at (455,260)-(486,281): text "2400"
rectangle at (455,290)-(486,311): text "2000"
rectangle at (455,320)-(486,341): text "1600"
rectangle at (455,350)-(486,371): text "1200"
rectangle at (455,380)-(486,401): text "800"
rectangle at (565,260)-(596,281): text "700"
rectangle at (565,290)-(596,311): text "575"
rectangle at (565,320)-(596,341): text "450"
rectangle at (565,350)-(596,371): text "325"
rectangle at (565,380)-(596,401): text "200"
rectangle at (50,140)-(121,161): text "READS"
rectangle at (780,105)-(861,126): text "%.1f s"; shows PARAMS.stDE601Cfg.TimeMax; runs INTERN ASSIGN INPUTS.PresSelCalStbd[9]:=(FALSE); editable
rectangle at (780,90)-(861,106): text "Time Max"
rectangle at (780,205)-(861,226): text "Dw: %.0f bar"; shows P601.MaxBar; runs INTERN ASSIGN INPUTS.PresSelCalStbd[9]:=(FALSE); editable
rectangle at (780,190)-(861,206): text "Press. Max"
rectangle at (780,145)-(861,166): text "Dw: %d"; shows PARAMS.stDE601Cfg.HP_Dw; runs INTERN ASSIGN INPUTS.PresSelCalStbd[9]:=(FALSE); editable 1..2
rectangle at (780,130)-(861,146): text "HP Pumps"
rectangle at (780,225)-(861,246): text "Up: %.0f bar"; shows P603.MaxBar; runs INTERN ASSIGN INPUTS.PresSelCalStbd[9]:=(FALSE); editable
rectangle at (780,165)-(861,186): text "Up: %d"; shows PARAMS.stDE601Cfg.HP_Up; runs INTERN ASSIGN INPUTS.PresSelCalStbd[9]:=(FALSE); editable 1..2
rectangle at (780,265)-(861,286): text "Dw: %.0f bar"; shows PARAMS.stDE601Cfg.TgtP_Dw; runs INTERN ASSIGN INPUTS.PresSelCalStbd[9]:=(FALSE); editable
rectangle at (780,250)-(861,266): text "TGT Press."
rectangle at (780,285)-(861,306): text "Up: %.0f bar"; shows PARAMS.stDE601Cfg.TgtP_Up; runs INTERN ASSIGN INPUTS.PresSelCalStbd[9]:=(FALSE); editable
rectangle at (780,310)-(861,331): text "DB: %.0f bar"; shows PARAMS.stDE601Cfg.P_DB; runs INTERN ASSIGN INPUTS.PresSelCalStbd[9]:=(FALSE); editable
rectangle at (780,350)-(861,371): text "Dw: %.0f %%"; shows PARAMS.stDE601Cfg.TgtLS_Dw; runs INTERN ASSIGN INPUTS.PresSelCalStbd[9]:=(FALSE); editable
rectangle at (780,335)-(861,351): text "TGT Pos."
rectangle at (780,370)-(861,391): text "Up: %.0f %%"; shows PARAMS.stDE601Cfg.TgtLS_Up; runs INTERN ASSIGN INPUTS.PresSelCalStbd[9]:=(FALSE); editable
rectangle at (780,435)-(861,456): text "Dw: %.1f s"; shows PARAMS.stDE601Cfg.Delay_Dw; runs INTERN ASSIGN INPUTS.PresSelCalStbd[9]:=(FALSE); editable
rectangle at (780,420)-(861,436): text "Time Push"
rectangle at (780,455)-(861,476): text "Up: %.1f s"; shows PARAMS.stDE601Cfg.Delay_Up; runs INTERN ASSIGN INPUTS.PresSelCalStbd[9]:=(FALSE); editable
rectangle at (780,395)-(861,416): text "DB: %.0f %%"; shows PARAMS.stDE601Cfg.LS_DB; runs INTERN ASSIGN INPUTS.PresSelCalStbd[9]:=(FALSE); editable
rectangle at (795,55)-(846,86): text "PROP. / UP/DW"
rounded rectangle at (90,505)-(141,526): text "RESET"; runs INTERN ASSIGN MAIN.Prop_UsedTime:=(0)
rectangle at (30,505)-(86,526): text "%.1f h"; shows MAIN.Prop_UsedTime / 3600; runs INTERN ASSIGN INPUTS.PresSelCalStbd[9]:=(FALSE)
rectangle at (30,490)-(86,506): text "Used Time"
rectangle at (525,455)-(591,476): text "Mild Temp."
rectangle at (590,455)-(661,476): text "%.0f °C"; shows S1100.LowDeg; runs INTERN ASSIGN INPUTS.PresSelCalStbd[9]:=(FALSE); editable
rectangle at (525,475)-(591,496): text "High Temp."
rectangle at (590,475)-(661,496): text "%.0f °C"; shows S1100.HigDeg; runs INTERN ASSIGN INPUTS.PresSelCalStbd[9]:=(FALSE); editable
rectangle at (525,495)-(591,516): text "Max. Temp."
rectangle at (590,495)-(661,516): text "%.0f °C"; shows S1100.MaxDeg; runs INTERN ASSIGN INPUTS.PresSelCalStbd[9]:=(FALSE); editable
rectangle at (300,445)-(351,466): text "RAW"
rectangle at (300,505)-(351,526): text "FINAL"
rectangle at (300,465)-(351,486): text "K"
rectangle at (300,485)-(351,506): text "OFF"
rectangle at (200,420)-(281,441): text "S1100 TEMP"
rectangle at (360,505)-(431,526): text "%.0f °C"; shows S1100.Deg
rectangle at (360,465)-(431,486): text "%.3f"; shows S1100.Cal_K; runs INTERN ASSIGN INPUTS.PresSelCalStbd[9]:=(FALSE); editable
rectangle at (360,445)-(431,466): text "%.3f V"; shows S1100.Raw; alarm colour if S1100.Err; runs INTERN ASSIGN INPUTS.PresSelCalStbd[9]:=(FALSE)
rectangle at (360,485)-(431,506): text "%.3f"; shows S1100.Cal_Off; runs INTERN ASSIGN INPUTS.PresSelCalStbd[9]:=(FALSE); editable
rectangle at (360,420)-(431,441): text "CALIB"
rectangle at (555,420)-(626,441): text "LIMITS"
290 more shapes without text or variables
*)

(* Visualisation VISU_CFG_SPECIAL
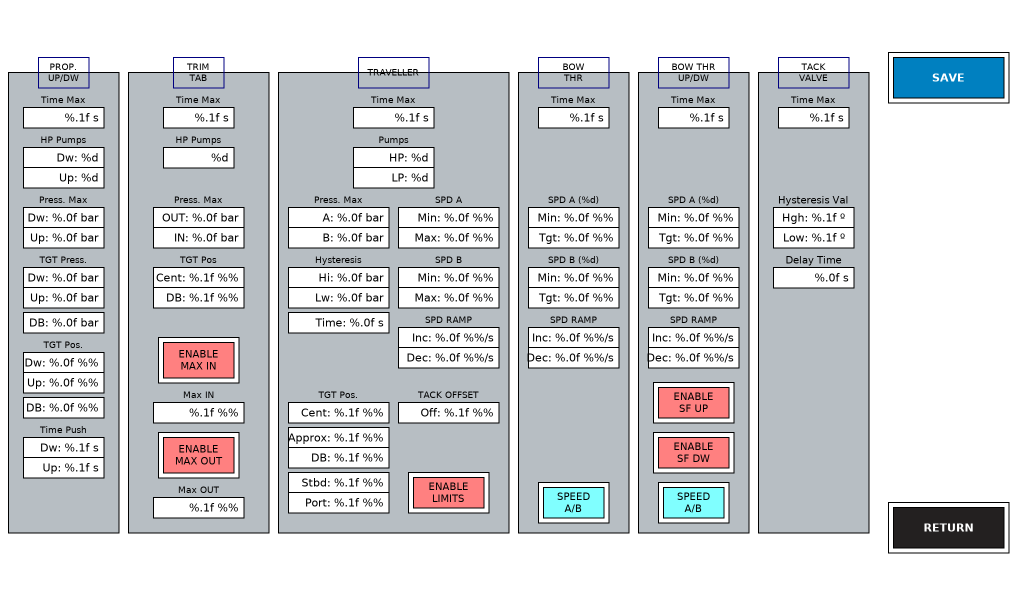
rectangle at (20,550)-(331,601): text "%s"; shows INPUTS.sVisuTime
rounded rectangle at (905,55)-(1016,96): text "SAVE"; alarm colour if PARAMS.Save; toggles PARAMS.Save
rounded rectangle at (905,505)-(1016,546): text "RETURN"; opens VISU_1_SPECIAL
rectangle at (730,550)-(896,601): text "SAVED!"; invisible if PARAMS.Saved
rectangle at (20,0)-(426,51): text "CFG: SPECIAL"
rectangle at (175,105)-(246,126): text "%.1f s"; shows PARAMS.stDE605Cfg.TimeMax; runs INTERN ASSIGN INPUTS.PresSelCalStbd[9]:=(FALSE); editable
rectangle at (165,400)-(256,421): text "%.1f %%"; shows PARAMS.stDE605Cfg.TgtLS_In; runs INTERN ASSIGN INPUTS.PresSelCalStbd[9]:=(FALSE); editable
rectangle at (175,90)-(246,106): text "Time Max"
rectangle at (175,385)-(246,401): text "Max IN"
rectangle at (165,205)-(256,226): text "OUT: %.0f bar"; shows P605.MaxBar; runs INTERN ASSIGN INPUTS.PresSelCalStbd[9]:=(FALSE); editable
rectangle at (175,190)-(246,206): text "Press. Max"
rectangle at (165,495)-(256,516): text "%.1f %%"; shows PARAMS.stDE605Cfg.TgtLS_Out; runs INTERN ASSIGN INPUTS.PresSelCalStbd[9]:=(FALSE); editable
rectangle at (175,480)-(246,496): text "Max OUT"
rectangle at (175,145)-(246,166): text "%d"; shows PARAMS.stDE605Cfg.HP; runs INTERN ASSIGN INPUTS.PresSelCalStbd[9]:=(FALSE); editable 1..2
rectangle at (175,130)-(246,146): text "HP Pumps"
rounded rectangle at (175,340)-(246,376): text "ENABLE / MAX IN"; alarm colour if PARAMS.stDE605Cfg.LS_Limit_In; toggles PARAMS.stDE605Cfg.LS_Limit_In
rounded rectangle at (175,435)-(246,471): text "ENABLE / MAX OUT"; alarm colour if PARAMS.stDE605Cfg.LS_Limit_Out; toggles PARAMS.stDE605Cfg.LS_Limit_Out
rectangle at (165,225)-(256,246): text "IN: %.0f bar"; shows P607.MaxBar; runs INTERN ASSIGN INPUTS.PresSelCalStbd[9]:=(FALSE); editable
rectangle at (165,265)-(256,286): text "Cent: %.1f %%"; shows PARAMS.stDE605Cfg.TgtLS_Mid; runs INTERN ASSIGN INPUTS.PresSelCalStbd[9]:=(FALSE); editable
rectangle at (175,250)-(246,266): text "TGT Pos"
rectangle at (165,285)-(256,306): text "DB: %.1f %%"; shows PARAMS.stDE605Cfg.TgtLS_DB; runs INTERN ASSIGN INPUTS.PresSelCalStbd[9]:=(FALSE); editable
rectangle at (35,105)-(116,126): text "%.1f s"; shows PARAMS.stDE601Cfg.TimeMax; runs INTERN ASSIGN INPUTS.PresSelCalStbd[9]:=(FALSE); editable
rectangle at (35,90)-(116,106): text "Time Max"
rectangle at (35,205)-(116,226): text "Dw: %.0f bar"; shows P601.MaxBar; runs INTERN ASSIGN INPUTS.PresSelCalStbd[9]:=(FALSE); editable
rectangle at (35,190)-(116,206): text "Press. Max"
rectangle at (35,145)-(116,166): text "Dw: %d"; shows PARAMS.stDE601Cfg.HP_Dw; runs INTERN ASSIGN INPUTS.PresSelCalStbd[9]:=(FALSE); editable 1..2
rectangle at (35,130)-(116,146): text "HP Pumps"
rectangle at (35,225)-(116,246): text "Up: %.0f bar"; shows P603.MaxBar; runs INTERN ASSIGN INPUTS.PresSelCalStbd[9]:=(FALSE); editable
rectangle at (35,165)-(116,186): text "Up: %d"; shows PARAMS.stDE601Cfg.HP_Up; runs INTERN ASSIGN INPUTS.PresSelCalStbd[9]:=(FALSE); editable 1..2
rectangle at (35,265)-(116,286): text "Dw: %.0f bar"; shows PARAMS.stDE601Cfg.TgtP_Dw; runs INTERN ASSIGN INPUTS.PresSelCalStbd[9]:=(FALSE); editable
rectangle at (35,250)-(116,266): text "TGT Press."
rectangle at (35,285)-(116,306): text "Up: %.0f bar"; shows PARAMS.stDE601Cfg.TgtP_Up; runs INTERN ASSIGN INPUTS.PresSelCalStbd[9]:=(FALSE); editable
rectangle at (35,310)-(116,331): text "DB: %.0f bar"; shows PARAMS.stDE601Cfg.P_DB; runs INTERN ASSIGN INPUTS.PresSelCalStbd[9]:=(FALSE); editable
rectangle at (35,350)-(116,371): text "Dw: %.0f %%"; shows PARAMS.stDE601Cfg.TgtLS_Dw; runs INTERN ASSIGN INPUTS.PresSelCalStbd[9]:=(FALSE); editable
rectangle at (35,335)-(116,351): text "TGT Pos."
rectangle at (35,370)-(116,391): text "Up: %.0f %%"; shows PARAMS.stDE601Cfg.TgtLS_Up; runs INTERN ASSIGN INPUTS.PresSelCalStbd[9]:=(FALSE); editable
rectangle at (35,435)-(116,456): text "Dw: %.1f s"; shows PARAMS.stDE601Cfg.Delay_Dw; runs INTERN ASSIGN INPUTS.PresSelCalStbd[9]:=(FALSE); editable
rectangle at (35,420)-(116,436): text "Time Push"
rectangle at (35,455)-(116,476): text "Up: %.1f s"; shows PARAMS.stDE601Cfg.Delay_Up; runs INTERN ASSIGN INPUTS.PresSelCalStbd[9]:=(FALSE); editable
rectangle at (35,395)-(116,416): text "DB: %.0f %%"; shows PARAMS.stDE601Cfg.LS_DB; runs INTERN ASSIGN INPUTS.PresSelCalStbd[9]:=(FALSE); editable
rectangle at (365,105)-(446,126): text "%.1f s"; shows PARAMS.stTravellerCfg.TimeMax; runs INTERN ASSIGN INPUTS.PresSelCalStbd[9]:=(FALSE); editable
rectangle at (300,470)-(401,491): text "Stbd: %.1f %%"; shows PARAMS.stTravellerCfg.TgtLS_Min; runs INTERN ASSIGN INPUTS.PresSelCalStbd[9]:=(FALSE); editable
rectangle at (365,90)-(446,106): text "Time Max"
rectangle at (300,205)-(401,226): text "A: %.0f bar"; shows P1301.MaxBar; runs INTERN ASSIGN INPUTS.PresSelCalStbd[9]:=(FALSE); editable
rectangle at (310,190)-(391,206): text "Press. Max"
rectangle at (300,490)-(401,511): text "Port: %.1f %%"; shows PARAMS.stTravellerCfg.TgtLS_Max; runs INTERN ASSIGN INPUTS.PresSelCalStbd[9]:=(FALSE); editable
rectangle at (365,145)-(446,166): text "HP: %d"; shows PARAMS.stTravellerCfg.HP; runs INTERN ASSIGN INPUTS.PresSelCalStbd[9]:=(FALSE); editable 1..2
rectangle at (365,130)-(446,146): text "Pumps"
rounded rectangle at (425,475)-(496,506): text "ENABLE / LIMITS"; alarm colour if PARAMS.stTravellerCfg.LS_Limit; toggles PARAMS.stTravellerCfg.LS_Limit
rectangle at (300,225)-(401,246): text "B: %.0f bar"; shows P1302.MaxBar; runs INTERN ASSIGN INPUTS.PresSelCalStbd[9]:=(FALSE); editable
rectangle at (300,400)-(401,421): text "Cent: %.1f %%"; shows PARAMS.stTravellerCfg.TgtLS_Zero; runs INTERN ASSIGN INPUTS.PresSelCalStbd[9]:=(FALSE); editable
rectangle at (310,385)-(391,401): text "TGT Pos."
rectangle at (300,425)-(401,446): text "Approx: %.1f %%"; shows PARAMS.stTravellerCfg.LS_Dist; runs INTERN ASSIGN INPUTS.PresSelCalStbd[9]:=(FALSE); editable
rectangle at (410,205)-(511,226): text "Min: %.0f %%"; shows PARAMS.stTravellerCfg.MinEVPA; runs INTERN ASSIGN INPUTS.PresSelCalStbd[9]:=(FALSE); editable
rectangle at (420,190)-(501,206): text "SPD A"
rectangle at (410,225)-(511,246): text "Max: %.0f %%"; shows PARAMS.stTravellerCfg.MaxEVPA; runs INTERN ASSIGN INPUTS.PresSelCalStbd[9]:=(FALSE); editable
rectangle at (410,265)-(511,286): text "Min: %.0f %%"; shows PARAMS.stTravellerCfg.MinEVPB; runs INTERN ASSIGN INPUTS.PresSelCalStbd[9]:=(FALSE); editable
rectangle at (420,250)-(501,266): text "SPD B"
rectangle at (410,285)-(511,306): text "Max: %.0f %%"; shows PARAMS.stTravellerCfg.MaxEVPB; runs INTERN ASSIGN INPUTS.PresSelCalStbd[9]:=(FALSE); editable
rectangle at (550,105)-(621,126): text "%.1f s"; shows PARAMS.stW1602Cfg.TimeMax; runs INTERN ASSIGN INPUTS.PresSelCalStbd[9]:=(FALSE); editable
rectangle at (540,205)-(631,226): text "Min: %.0f %%"; shows PARAMS.stBowThrCfg.SpdA_Min; runs INTERN ASSIGN INPUTS.PresSelCalStbd[9]:=(FALSE); editable
rectangle at (550,90)-(621,106): text "Time Max"
rectangle at (550,190)-(621,206): text "SPD A (%d)"; shows MAIN.fbBowThr.SpdA
rectangle at (540,265)-(631,286): text "Min: %.0f %%"; shows PARAMS.stBowThrCfg.SpdB_Min; runs INTERN ASSIGN INPUTS.PresSelCalStbd[9]:=(FALSE); editable
rounded rectangle at (555,485)-(616,516): text "SPEED / A/B"; toggles PARAMS.stBowThrCfg.A_Spd1
rectangle at (550,250)-(621,266): text "SPD B (%d)"; shows MAIN.fbBowThr.SpdB
rectangle at (670,105)-(741,126): text "%.1f s"; shows PARAMS.stW1604Cfg.TimeMax; runs INTERN ASSIGN INPUTS.PresSelCalStbd[9]:=(FALSE); editable
rectangle at (660,205)-(751,226): text "Min: %.0f %%"; shows PARAMS.stBowThrUpDwCfg.SpdA_Min; runs INTERN ASSIGN INPUTS.PresSelCalStbd[9]:=(FALSE); editable
rectangle at (670,90)-(741,106): text "Time Max"
rectangle at (670,190)-(741,206): text "SPD A (%d)"; shows MAIN.fbBowThrUpDw.SpdA
rectangle at (660,265)-(751,286): text "Min: %.0f %%"; shows PARAMS.stBowThrUpDwCfg.SpdB_Min; runs INTERN ASSIGN INPUTS.PresSelCalStbd[9]:=(FALSE); editable
rounded rectangle at (675,485)-(736,516): text "SPEED / A/B"; toggles PARAMS.stBowThrUpDwCfg.A_Spd1
rectangle at (670,250)-(741,266): text "SPD B (%d)"; shows MAIN.fbBowThrUpDw.SpdB
rectangle at (300,445)-(401,466): text "DB: %.1f %%"; shows PARAMS.stTravellerCfg.LS_DB; runs INTERN ASSIGN INPUTS.PresSelCalStbd[9]:=(FALSE); editable
rounded rectangle at (670,435)-(741,466): text "ENABLE / SF DW"; alarm colour if PARAMS.stBowThrUpDwCfg.SF2_Limit; toggles PARAMS.stBowThrUpDwCfg.SF2_Limit
rounded rectangle at (670,385)-(741,416): text "ENABLE / SF UP"; alarm colour if PARAMS.stBowThrUpDwCfg.SF1_Limit; toggles PARAMS.stBowThrUpDwCfg.SF1_Limit
rectangle at (660,225)-(751,246): text "Tgt: %.0f %%"; shows PARAMS.stBowThrUpDwCfg.SpdA_Max; runs INTERN ASSIGN INPUTS.PresSelCalStbd[9]:=(FALSE); editable
rectangle at (540,225)-(631,246): text "Tgt: %.0f %%"; shows PARAMS.stBowThrCfg.SpdA_Max; runs INTERN ASSIGN INPUTS.PresSelCalStbd[9]:=(FALSE); editable
rectangle at (540,285)-(631,306): text "Tgt: %.0f %%"; shows PARAMS.stBowThrCfg.SpdB_Max; runs INTERN ASSIGN INPUTS.PresSelCalStbd[9]:=(FALSE); editable
rectangle at (660,285)-(751,306): text "Tgt: %.0f %%"; shows PARAMS.stBowThrUpDwCfg.SpdB_Max; runs INTERN ASSIGN INPUTS.PresSelCalStbd[9]:=(FALSE); editable
rectangle at (540,325)-(631,346): text "Inc: %.0f %%/s"; shows PARAMS.stBowThrCfg.Spd_Inc; runs INTERN ASSIGN INPUTS.PresSelCalStbd[9]:=(FALSE); editable
rectangle at (550,310)-(621,326): text "SPD RAMP"; shows MAIN.fbW1602.SpdA
rectangle at (660,325)-(751,346): text "Inc: %.0f %%/s"; shows PARAMS.stBowThrUpDwCfg.Spd_Inc; runs INTERN ASSIGN INPUTS.PresSelCalStbd[9]:=(FALSE); editable
rectangle at (670,310)-(741,326): text "SPD RAMP"; shows MAIN.fbW1604.SpdA
rectangle at (660,345)-(751,366): text "Dec: %.0f %%/s"; shows PARAMS.stBowThrUpDwCfg.Spd_Dec; runs INTERN ASSIGN INPUTS.PresSelCalStbd[9]:=(FALSE); editable
rectangle at (540,345)-(631,366): text "Dec: %.0f %%/s"; shows PARAMS.stBowThrCfg.Spd_Dec; runs INTERN ASSIGN INPUTS.PresSelCalStbd[9]:=(FALSE); editable
rectangle at (410,325)-(511,346): text "Inc: %.0f %%/s"; shows PARAMS.stTravellerCfg.Spd_Inc; runs INTERN ASSIGN INPUTS.PresSelCalStbd[9]:=(FALSE); editable
rectangle at (425,310)-(496,326): text "SPD RAMP"; shows MAIN.fbW1604.SpdA
rectangle at (410,345)-(511,366): text "Dec: %.0f %%/s"; shows PARAMS.stTravellerCfg.Spd_Dec; runs INTERN ASSIGN INPUTS.PresSelCalStbd[9]:=(FALSE); editable
rectangle at (365,165)-(446,186): text "LP: %d"; shows PARAMS.stTravellerCfg.LP; runs INTERN ASSIGN INPUTS.PresSelCalStbd[9]:=(FALSE); editable 1..2
rectangle at (300,265)-(401,286): text "Hi: %.0f bar"; shows PARAMS.stTravellerCfg.Hyst_HP; runs INTERN ASSIGN INPUTS.PresSelCalStbd[9]:=(FALSE); editable
rectangle at (300,285)-(401,306): text "Lw: %.0f bar"; shows PARAMS.stTravellerCfg.Hyst_LP; runs INTERN ASSIGN INPUTS.PresSelCalStbd[9]:=(FALSE); editable
rectangle at (300,310)-(401,331): text "Time: %.0f s"; shows PARAMS.stTravellerCfg.Hyst_TM; runs INTERN ASSIGN INPUTS.PresSelCalStbd[9]:=(FALSE); editable
rectangle at (310,250)-(391,266): text "Hysteresis"
rectangle at (410,400)-(511,421): text "Off: %.1f %%"; shows PARAMS.stTravellerCfg.TgtLS_Tack_Off; runs INTERN ASSIGN INPUTS.PresSelCalStbd[9]:=(FALSE); editable
rectangle at (410,385)-(511,401): text "TACK OFFSET"
rectangle at (185,55)-(236,86): text "TRIM / TAB"
rectangle at (50,55)-(101,86): text "PROP. / UP/DW"
rectangle at (370,55)-(441,86): text "TRAVELLER"
rectangle at (550,55)-(621,86): text "BOW / THR"
rectangle at (670,55)-(741,86): text "BOW THR / UP/DW"
rectangle at (790,55)-(861,86): text "TACK / VALVE"
rectangle at (790,105)-(861,126): text "%.1f s"; shows PARAMS.stTackValveCfg.TimeMax; runs INTERN ASSIGN INPUTS.PresSelCalStbd[9]:=(FALSE); editable
rectangle at (790,90)-(861,106): text "Time Max"
rectangle at (785,205)-(866,226): text "Hgh: %.1f º"; shows PARAMS.stTackValveCfg.Hyst_HeelH; runs INTERN ASSIGN INPUTS.PresSelCalStbd[9]:=(FALSE); editable
rectangle at (785,225)-(866,246): text "Low: %.1f º"; shows PARAMS.stTackValveCfg.Hyst_HeelL; runs INTERN ASSIGN INPUTS.PresSelCalStbd[9]:=(FALSE); editable
rectangle at (785,265)-(866,286): text "%.0f s"; shows PARAMS.stTackValveCfg.Hyst_Time; runs INTERN ASSIGN INPUTS.PresSelCalStbd[9]:=(FALSE); editable
rectangle at (780,190)-(871,206): text "Hysteresis Val"; shows RECV_J1939.F004.DriverDemandTorque
rectangle at (780,250)-(871,266): text "Delay Time"; shows RECV_J1939.F004.DriverDemandTorque
15 more shapes without text or variables
*)

(* Visualisation VISU_CFG_TANK
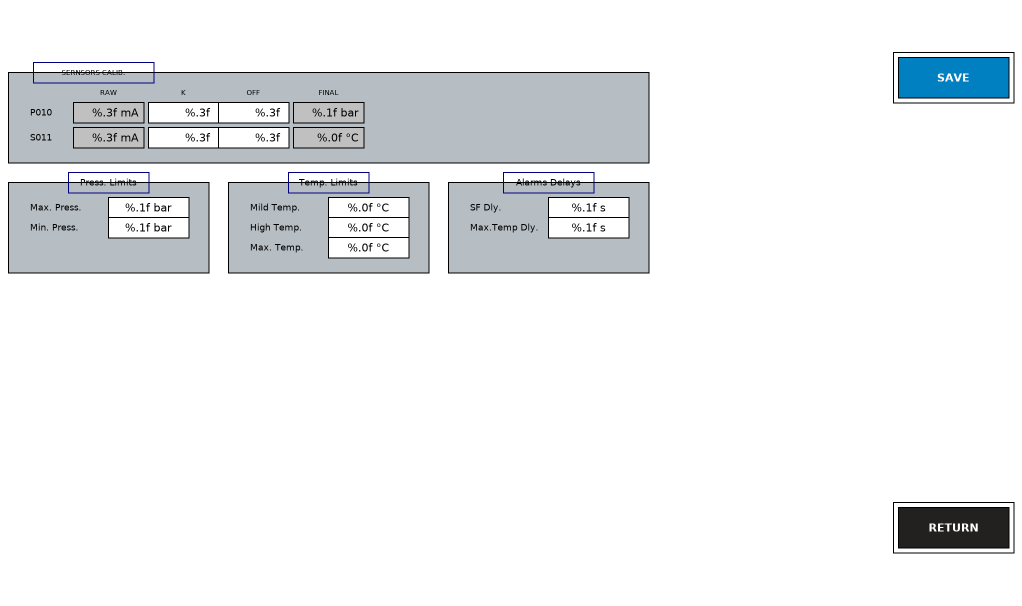
rectangle at (20,0)-(331,51): text "CFG: TANK"
rectangle at (35,100)-(81,121): text "P010"
rectangle at (80,80)-(151,101): text "RAW"
rectangle at (300,100)-(371,121): text "%.1f bar"; shows P010.Bar
rectangle at (155,100)-(226,121): text "%.3f"; shows P010.Cal_K; runs INTERN ASSIGN INPUTS.PresSelCalStbd[9]:=(FALSE); editable
rectangle at (80,100)-(151,121): text "%.3f mA"; shows P010.Raw; alarm colour if P010.Err; runs INTERN ASSIGN INPUTS.PresSelCalStbd[9]:=(FALSE)
rectangle at (225,100)-(296,121): text "%.3f"; shows P010.Cal_Off; runs INTERN ASSIGN INPUTS.PresSelCalStbd[9]:=(FALSE); editable
rectangle at (300,80)-(371,101): text "FINAL"
rectangle at (155,80)-(226,101): text "K"
rectangle at (225,80)-(296,101): text "OFF"
rectangle at (20,550)-(331,601): text "%s"; shows INPUTS.sVisuTime
rectangle at (40,60)-(161,81): text "SERNSORS CALIB."
rectangle at (35,195)-(116,216): text "Max. Press."
rectangle at (115,195)-(196,216): text "%.1f bar"; shows P010.MaxBar; runs INTERN ASSIGN INPUTS.PresSelCalStbd[9]:=(FALSE); editable
rectangle at (35,215)-(116,236): text "Min. Press."
rectangle at (115,215)-(196,236): text "%.1f bar"; shows P010.MinBar; runs INTERN ASSIGN INPUTS.PresSelCalStbd[9]:=(FALSE); editable
rectangle at (75,170)-(156,191): text "Press. Limits"
rectangle at (475,195)-(556,216): text "SF Dly."
rectangle at (555,195)-(636,216): text "%.1f s"; shows PARAMS.SF_Delay; runs INTERN ASSIGN INPUTS.PresSelCalStbd[9]:=(FALSE); editable
rectangle at (510,170)-(601,191): text "Alarms Delays"
rounded rectangle at (905,55)-(1016,96): text "SAVE"; alarm colour if PARAMS.Save; toggles PARAMS.Save
rounded rectangle at (905,505)-(1016,546): text "RETURN"; opens VISU_1_TANK
rectangle at (35,125)-(81,146): text "S011"
rectangle at (300,125)-(371,146): text "%.0f °C"; shows S011.Deg
rectangle at (155,125)-(226,146): text "%.3f"; shows S011.Cal_K; runs INTERN ASSIGN INPUTS.PresSelCalStbd[9]:=(FALSE); editable
rectangle at (80,125)-(151,146): text "%.3f mA"; shows S011.Raw; alarm colour if S011.Err; runs INTERN ASSIGN INPUTS.PresSelCalStbd[9]:=(FALSE)
rectangle at (225,125)-(296,146): text "%.3f"; shows S011.Cal_Off; runs INTERN ASSIGN INPUTS.PresSelCalStbd[9]:=(FALSE); editable
rectangle at (255,195)-(336,216): text "Mild Temp."
rectangle at (335,195)-(416,216): text "%.0f °C"; shows S011.LowDeg; runs INTERN ASSIGN INPUTS.PresSelCalStbd[9]:=(FALSE); editable
rectangle at (255,215)-(336,236): text "High Temp."
rectangle at (335,215)-(416,236): text "%.0f °C"; shows S011.HigDeg; runs INTERN ASSIGN INPUTS.PresSelCalStbd[9]:=(FALSE); editable
rectangle at (295,170)-(376,191): text "Temp. Limits"
rectangle at (255,235)-(336,256): text "Max. Temp."
rectangle at (335,235)-(416,256): text "%.0f °C"; shows S011.MaxDeg; runs INTERN ASSIGN INPUTS.PresSelCalStbd[9]:=(FALSE); editable
rectangle at (475,215)-(556,236): text "Max.Temp Dly."
rectangle at (555,215)-(636,236): text "%.1f s"; shows S011.Delay; runs INTERN ASSIGN INPUTS.PresSelCalStbd[9]:=(FALSE); editable
rectangle at (730,550)-(896,601): text "SAVED!"; invisible if PARAMS.Saved
6 more shapes without text or variables
*)

(* Visualisation VISU_CFG_WB
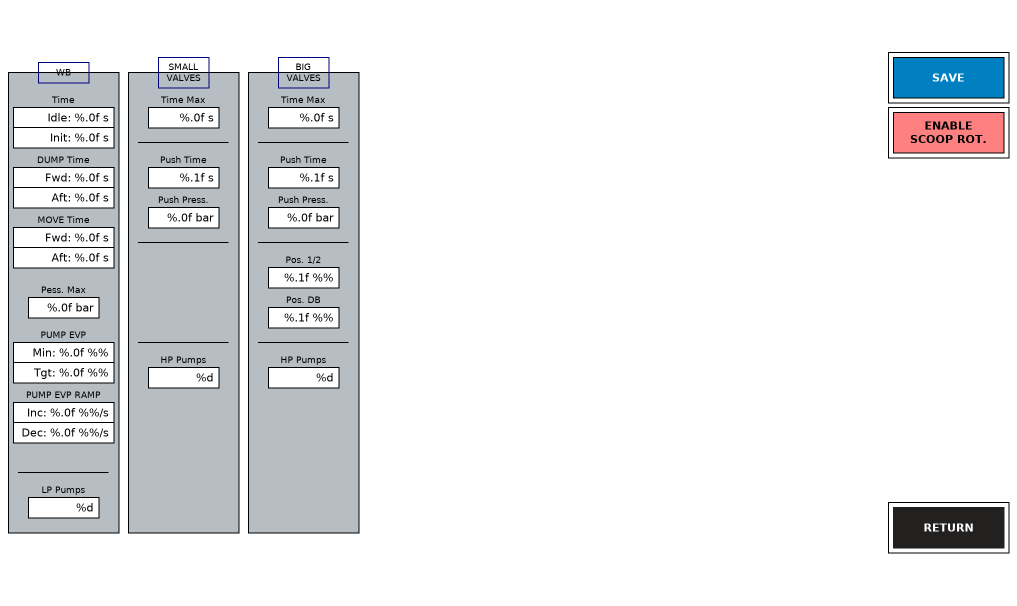
rectangle at (20,550)-(331,601): text "%s"; shows INPUTS.sVisuTime
rounded rectangle at (905,55)-(1016,96): text "SAVE"; alarm colour if PARAMS.Save; toggles PARAMS.Save
rounded rectangle at (905,505)-(1016,546): text "RETURN"; opens VISU_1_WB
rectangle at (730,550)-(896,601): text "SAVED!"; invisible if PARAMS.Saved
rectangle at (160,90)-(231,106): text "Time Max"
rectangle at (160,190)-(231,206): text "Push Press."
rectangle at (170,55)-(221,86): text "SMALL / VALVES"
rectangle at (290,55)-(341,86): text "BIG / VALVES"
rectangle at (160,165)-(231,186): text "%.1f s"; shows PARAMS.stWBValveSFCfg.PushTime; runs INTERN ASSIGN INPUTS.PresSelCalStbd[9]:=(FALSE); editable
rectangle at (160,150)-(231,166): text "Push Time"
rectangle at (160,365)-(231,386): text "%d"; shows PARAMS.stWBValveSFCfg.HP; runs INTERN ASSIGN INPUTS.PresSelCalStbd[9]:=(FALSE); editable 1..2
rectangle at (160,350)-(231,366): text "HP Pumps"
rectangle at (280,265)-(351,286): text "%.1f %%"; shows PARAMS.stWBValveLSCfg.TgtLS_Half; runs INTERN ASSIGN INPUTS.PresSelCalStbd[9]:=(FALSE); editable
rectangle at (280,90)-(351,106): text "Time Max"
rectangle at (280,250)-(351,266): text "Pos. 1/2"
rectangle at (280,305)-(351,326): text "%.1f %%"; shows PARAMS.stWBValveLSCfg.LS_DB; runs INTERN ASSIGN INPUTS.PresSelCalStbd[9]:=(FALSE); editable
rectangle at (280,290)-(351,306): text "Pos. DB"
rectangle at (20,0)-(426,51): text "CFG: WATER BALLAST"
rectangle at (160,105)-(231,126): text "%.0f s"; shows PARAMS.stWBValveSFCfg.TimeMax; runs INTERN ASSIGN INPUTS.PresSelCalStbd[9]:=(FALSE); editable
rectangle at (280,105)-(351,126): text "%.0f s"; shows PARAMS.stWBValveLSCfg.TimeMax; runs INTERN ASSIGN INPUTS.PresSelCalStbd[9]:=(FALSE); editable
rectangle at (160,205)-(231,226): text "%.0f bar"; shows PARAMS.stWBValveSFCfg.PushP; runs INTERN ASSIGN INPUTS.PresSelCalStbd[9]:=(FALSE); editable
rectangle at (280,190)-(351,206): text "Push Press."
rectangle at (280,165)-(351,186): text "%.1f s"; shows PARAMS.stWBValveLSCfg.PushTime; runs INTERN ASSIGN INPUTS.PresSelCalStbd[9]:=(FALSE); editable
rectangle at (280,150)-(351,166): text "Push Time"
rectangle at (280,205)-(351,226): text "%.0f bar"; shows PARAMS.stWBValveLSCfg.PushP; runs INTERN ASSIGN INPUTS.PresSelCalStbd[9]:=(FALSE); editable
rectangle at (280,365)-(351,386): text "%d"; shows PARAMS.stWBValveLSCfg.HP; runs INTERN ASSIGN INPUTS.PresSelCalStbd[9]:=(FALSE); editable 1..2
rectangle at (280,350)-(351,366): text "HP Pumps"
rectangle at (40,280)-(111,296): text "Pess. Max"
rectangle at (40,295)-(111,316): text "%.0f bar"; shows P2500.MaxBar; runs INTERN ASSIGN INPUTS.PresSelCalStbd[9]:=(FALSE); editable
rectangle at (50,60)-(101,81): text "WB"
rectangle at (40,90)-(111,106): text "Time"
rectangle at (40,495)-(111,516): text "%d"; shows PARAMS.stWBCfg.LP; runs INTERN ASSIGN INPUTS.PresSelCalStbd[9]:=(FALSE); editable 1..2
rectangle at (40,480)-(111,496): text "LP Pumps"
rectangle at (25,340)-(126,361): text "Min: %.0f %%"; shows PARAMS.stWBCfg.EVP_Pump_Min; runs INTERN ASSIGN INPUTS.PresSelCalStbd[9]:=(FALSE); editable
rectangle at (25,360)-(126,381): text "Tgt: %.0f %%"; shows PARAMS.stWBCfg.EVP_Pump_Max; runs INTERN ASSIGN INPUTS.PresSelCalStbd[9]:=(FALSE); editable
rectangle at (40,325)-(111,341): text "PUMP EVP"
rectangle at (25,400)-(126,421): text "Inc: %.0f %%/s"; shows PARAMS.stWBCfg.EVP_Pump_Inc; runs INTERN ASSIGN INPUTS.PresSelCalStbd[9]:=(FALSE); editable
rectangle at (25,420)-(126,441): text "Dec: %.0f %%/s"; shows PARAMS.stWBCfg.EVP_Pump_Dec; runs INTERN ASSIGN INPUTS.PresSelCalStbd[9]:=(FALSE); editable
rectangle at (25,385)-(126,401): text "PUMP EVP RAMP"
rectangle at (25,105)-(126,126): text "Idle: %.0f s"; shows PARAMS.stWBCfg.TimeMax_Idle; runs INTERN ASSIGN INPUTS.PresSelCalStbd[9]:=(FALSE); editable
rectangle at (25,125)-(126,146): text "Init: %.0f s"; shows PARAMS.stWBCfg.TimeMax_Init; runs INTERN ASSIGN INPUTS.PresSelCalStbd[9]:=(FALSE); editable
rectangle at (25,165)-(126,186): text "Fwd: %.0f s"; shows PARAMS.stWBCfg.TimeMax_DumpFwd; runs INTERN ASSIGN INPUTS.PresSelCalStbd[9]:=(FALSE); editable
rectangle at (40,150)-(111,166): text "DUMP Time"
rectangle at (25,185)-(126,206): text "Aft: %.0f s"; shows PARAMS.stWBCfg.TimeMax_DumpAft; runs INTERN ASSIGN INPUTS.PresSelCalStbd[9]:=(FALSE); editable
rectangle at (25,225)-(126,246): text "Fwd: %.0f s"; shows PARAMS.stWBCfg.TimeMax_MoveFwd; runs INTERN ASSIGN INPUTS.PresSelCalStbd[9]:=(FALSE); editable
rectangle at (40,210)-(111,226): text "MOVE Time"
rectangle at (25,245)-(126,266): text "Aft: %.0f s"; shows PARAMS.stWBCfg.TimeMax_MoveAft; runs INTERN ASSIGN INPUTS.PresSelCalStbd[9]:=(FALSE); editable
rounded rectangle at (905,110)-(1016,151): text "ENABLE / SCOOP ROT."; alarm colour if PARAMS.stWBCfg.EnScoopAF; toggles PARAMS.stWBCfg.EnScoopAF
13 more shapes without text or variables
*)

(* Visualisation VISU_CFG_WINCHES
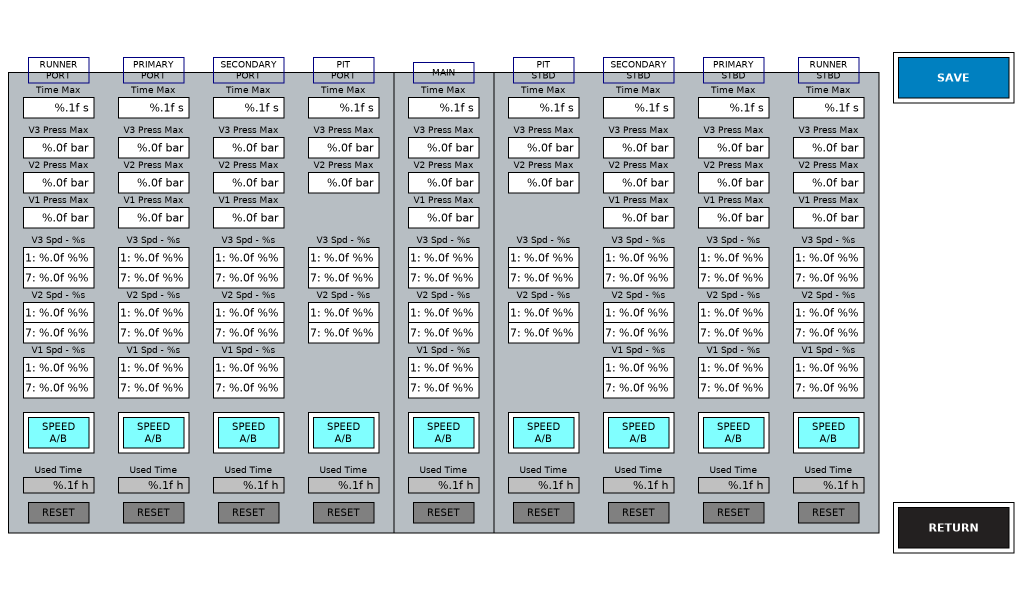
rectangle at (20,0)-(426,51): text "CFG: WINCHES"
rectangle at (20,550)-(331,601): text "%s"; shows INPUTS.sVisuTime
rounded rectangle at (905,55)-(1016,96): text "SAVE"; alarm colour if PARAMS.Save; toggles PARAMS.Save
rounded rectangle at (905,505)-(1016,546): text "RETURN"; opens VISU_1_WINCHES
rectangle at (705,95)-(776,116): text "%.1f s"; shows PARAMS.stW1202Cfg.TimeMax; runs INTERN ASSIGN INPUTS.PresSelCalStbd[9]:=(FALSE); editable
rectangle at (705,245)-(776,266): text "1: %.0f %%"; shows PARAMS.stW1202Cfg.Spd1[1]; runs INTERN ASSIGN INPUTS.PresSelCalStbd[9]:=(FALSE); editable
rectangle at (705,230)-(776,246): text "V3 Spd - %s"; shows MAIN.fbW1202.Spd1
rectangle at (705,300)-(776,321): text "1: %.0f %%"; shows PARAMS.stW1202Cfg.Spd2[1]; runs INTERN ASSIGN INPUTS.PresSelCalStbd[9]:=(FALSE); editable
rectangle at (705,320)-(776,341): text "7: %.0f %%"; shows PARAMS.stW1202Cfg.Spd2[7]; runs INTERN ASSIGN INPUTS.PresSelCalStbd[9]:=(FALSE); editable
rounded rectangle at (710,415)-(771,446): text "SPEED / A/B"; toggles PARAMS.stW1202Cfg.A_Spd1
rectangle at (705,285)-(776,301): text "V2 Spd - %s"; shows MAIN.fbW1202.Spd2
rectangle at (730,550)-(896,601): text "SAVED!"; invisible if PARAMS.Saved
rectangle at (515,95)-(586,116): text "%.1f s"; shows PARAMS.stW1204Cfg.TimeMax; runs INTERN ASSIGN INPUTS.PresSelCalStbd[9]:=(FALSE); editable
rectangle at (515,245)-(586,266): text "1: %.0f %%"; shows PARAMS.stW1204Cfg.Spd1[1]; runs INTERN ASSIGN INPUTS.PresSelCalStbd[9]:=(FALSE); editable
rectangle at (515,230)-(586,246): text "V3 Spd - %s"; shows MAIN.fbW1204.Spd1
rectangle at (515,300)-(586,321): text "1: %.0f %%"; shows PARAMS.stW1204Cfg.Spd2[1]; runs INTERN ASSIGN INPUTS.PresSelCalStbd[9]:=(FALSE); editable
rectangle at (515,320)-(586,341): text "7: %.0f %%"; shows PARAMS.stW1204Cfg.Spd2[7]; runs INTERN ASSIGN INPUTS.PresSelCalStbd[9]:=(FALSE); editable
rounded rectangle at (520,415)-(581,446): text "SPEED / A/B"; toggles PARAMS.stW1204Cfg.A_Spd1
rectangle at (515,285)-(586,301): text "V2 Spd - %s"; shows MAIN.fbW1204.Spd2
rectangle at (705,265)-(776,286): text "7: %.0f %%"; shows PARAMS.stW1202Cfg.Spd1[7]; runs INTERN ASSIGN INPUTS.PresSelCalStbd[9]:=(FALSE); editable
rectangle at (515,265)-(586,286): text "7: %.0f %%"; shows PARAMS.stW1204Cfg.Spd1[7]; runs INTERN ASSIGN INPUTS.PresSelCalStbd[9]:=(FALSE); editable
rectangle at (415,95)-(486,116): text "%.1f s"; shows PARAMS.stW1206Cfg.TimeMax; runs INTERN ASSIGN INPUTS.PresSelCalStbd[9]:=(FALSE); editable
rectangle at (415,245)-(486,266): text "1: %.0f %%"; shows PARAMS.stW1206Cfg.Spd1[1]; runs INTERN ASSIGN INPUTS.PresSelCalStbd[9]:=(FALSE); editable
rectangle at (415,230)-(486,246): text "V3 Spd - %s"; shows MAIN.fbW1206.Spd1
rectangle at (415,300)-(486,321): text "1: %.0f %%"; shows PARAMS.stW1206Cfg.Spd2[1]; runs INTERN ASSIGN INPUTS.PresSelCalStbd[9]:=(FALSE); editable
rectangle at (415,320)-(486,341): text "7: %.0f %%"; shows PARAMS.stW1206Cfg.Spd2[7]; runs INTERN ASSIGN INPUTS.PresSelCalStbd[9]:=(FALSE); editable
rounded rectangle at (420,415)-(481,446): text "SPEED / A/B"; toggles PARAMS.stW1206Cfg.A_Spd1
rectangle at (415,285)-(486,301): text "V2 Spd - %s"; shows MAIN.fbW1206.Spd2
rectangle at (30,95)-(101,116): text "%.1f s"; shows PARAMS.stW1208Cfg.TimeMax; runs INTERN ASSIGN INPUTS.PresSelCalStbd[9]:=(FALSE); editable
rectangle at (30,245)-(101,266): text "1: %.0f %%"; shows PARAMS.stW1208Cfg.Spd1[1]; runs INTERN ASSIGN INPUTS.PresSelCalStbd[9]:=(FALSE); editable
rectangle at (30,80)-(101,96): text "Time Max"
rectangle at (30,230)-(101,246): text "V3 Spd - %s"; shows MAIN.fbW1208.Spd1
rectangle at (30,300)-(101,321): text "1: %.0f %%"; shows PARAMS.stW1208Cfg.Spd2[1]; runs INTERN ASSIGN INPUTS.PresSelCalStbd[9]:=(FALSE); editable
rectangle at (30,320)-(101,341): text "7: %.0f %%"; shows PARAMS.stW1208Cfg.Spd2[7]; runs INTERN ASSIGN INPUTS.PresSelCalStbd[9]:=(FALSE); editable
rounded rectangle at (35,415)-(96,446): text "SPEED / A/B"; toggles PARAMS.stW1208Cfg.A_Spd1
rectangle at (30,285)-(101,301): text "V2 Spd - %s"; shows MAIN.fbW1208.Spd2
rectangle at (415,265)-(486,286): text "7: %.0f %%"; shows PARAMS.stW1206Cfg.Spd1[7]; runs INTERN ASSIGN INPUTS.PresSelCalStbd[9]:=(FALSE); editable
rectangle at (30,265)-(101,286): text "7: %.0f %%"; shows PARAMS.stW1208Cfg.Spd1[7]; runs INTERN ASSIGN INPUTS.PresSelCalStbd[9]:=(FALSE); editable
rectangle at (800,95)-(871,116): text "%.1f s"; shows PARAMS.stW1602Cfg.TimeMax; runs INTERN ASSIGN INPUTS.PresSelCalStbd[9]:=(FALSE); editable
rectangle at (800,245)-(871,266): text "1: %.0f %%"; shows PARAMS.stW1602Cfg.Spd1[1]; runs INTERN ASSIGN INPUTS.PresSelCalStbd[9]:=(FALSE); editable
rectangle at (800,230)-(871,246): text "V3 Spd - %s"; shows MAIN.fbW1602.Spd1
rectangle at (800,300)-(871,321): text "1: %.0f %%"; shows PARAMS.stW1602Cfg.Spd2[1]; runs INTERN ASSIGN INPUTS.PresSelCalStbd[9]:=(FALSE); editable
rectangle at (800,320)-(871,341): text "7: %.0f %%"; shows PARAMS.stW1602Cfg.Spd2[7]; runs INTERN ASSIGN INPUTS.PresSelCalStbd[9]:=(FALSE); editable
rounded rectangle at (805,415)-(866,446): text "SPEED / A/B"; toggles PARAMS.stW1602Cfg.A_Spd1
rectangle at (800,285)-(871,301): text "V2 Spd - %s"; shows MAIN.fbW1602.Spd2
rectangle at (610,95)-(681,116): text "%.1f s"; shows PARAMS.stW1604Cfg.TimeMax; runs INTERN ASSIGN INPUTS.PresSelCalStbd[9]:=(FALSE); editable
rectangle at (610,245)-(681,266): text "1: %.0f %%"; shows PARAMS.stW1604Cfg.Spd1[1]; runs INTERN ASSIGN INPUTS.PresSelCalStbd[9]:=(FALSE); editable
rectangle at (610,230)-(681,246): text "V3 Spd - %s"; shows MAIN.fbW1604.Spd1
rectangle at (610,300)-(681,321): text "1: %.0f %%"; shows PARAMS.stW1604Cfg.Spd2[1]; runs INTERN ASSIGN INPUTS.PresSelCalStbd[9]:=(FALSE); editable
rectangle at (610,320)-(681,341): text "7: %.0f %%"; shows PARAMS.stW1604Cfg.Spd2[7]; runs INTERN ASSIGN INPUTS.PresSelCalStbd[9]:=(FALSE); editable
rounded rectangle at (615,415)-(676,446): text "SPEED / A/B"; toggles PARAMS.stW1604Cfg.A_Spd1
rectangle at (610,285)-(681,301): text "V2 Spd - %s"; shows MAIN.fbW1604.Spd2
rectangle at (800,265)-(871,286): text "7: %.0f %%"; shows PARAMS.stW1602Cfg.Spd1[7]; runs INTERN ASSIGN INPUTS.PresSelCalStbd[9]:=(FALSE); editable
rectangle at (610,265)-(681,286): text "7: %.0f %%"; shows PARAMS.stW1604Cfg.Spd1[7]; runs INTERN ASSIGN INPUTS.PresSelCalStbd[9]:=(FALSE); editable
rectangle at (220,95)-(291,116): text "%.1f s"; shows PARAMS.stW1212Cfg.TimeMax; runs INTERN ASSIGN INPUTS.PresSelCalStbd[9]:=(FALSE); editable
rectangle at (220,245)-(291,266): text "1: %.0f %%"; shows PARAMS.stW1212Cfg.Spd1[1]; runs INTERN ASSIGN INPUTS.PresSelCalStbd[9]:=(FALSE); editable
rectangle at (220,230)-(291,246): text "V3 Spd - %s"; shows MAIN.fbW1212.Spd1
rectangle at (220,300)-(291,321): text "1: %.0f %%"; shows PARAMS.stW1212Cfg.Spd2[1]; runs INTERN ASSIGN INPUTS.PresSelCalStbd[9]:=(FALSE); editable
rectangle at (220,320)-(291,341): text "7: %.0f %%"; shows PARAMS.stW1212Cfg.Spd2[7]; runs INTERN ASSIGN INPUTS.PresSelCalStbd[9]:=(FALSE); editable
rounded rectangle at (225,415)-(286,446): text "SPEED / A/B"; toggles PARAMS.stW1212Cfg.A_Spd1
rectangle at (220,285)-(291,301): text "V2 Spd - %s"; shows MAIN.fbW1212.Spd2
rectangle at (315,95)-(386,116): text "%.1f s"; shows PARAMS.stW1214Cfg.TimeMax; runs INTERN ASSIGN INPUTS.PresSelCalStbd[9]:=(FALSE); editable
rectangle at (315,245)-(386,266): text "1: %.0f %%"; shows PARAMS.stW1214Cfg.Spd1[1]; runs INTERN ASSIGN INPUTS.PresSelCalStbd[9]:=(FALSE); editable
rectangle at (315,230)-(386,246): text "V3 Spd - %s"; shows MAIN.fbW1214.Spd1
rectangle at (315,300)-(386,321): text "1: %.0f %%"; shows PARAMS.stW1214Cfg.Spd2[1]; runs INTERN ASSIGN INPUTS.PresSelCalStbd[9]:=(FALSE); editable
rectangle at (315,320)-(386,341): text "7: %.0f %%"; shows PARAMS.stW1214Cfg.Spd2[7]; runs INTERN ASSIGN INPUTS.PresSelCalStbd[9]:=(FALSE); editable
rounded rectangle at (320,415)-(381,446): text "SPEED / A/B"; toggles PARAMS.stW1214Cfg.A_Spd1
rectangle at (315,285)-(386,301): text "V2 Spd - %s"; shows MAIN.fbW1214.Spd2
rectangle at (220,265)-(291,286): text "7: %.0f %%"; shows PARAMS.stW1212Cfg.Spd1[7]; runs INTERN ASSIGN INPUTS.PresSelCalStbd[9]:=(FALSE); editable
rectangle at (315,265)-(386,286): text "7: %.0f %%"; shows PARAMS.stW1214Cfg.Spd1[7]; runs INTERN ASSIGN INPUTS.PresSelCalStbd[9]:=(FALSE); editable
rectangle at (125,95)-(196,116): text "%.1f s"; shows PARAMS.stW1210Cfg.TimeMax; runs INTERN ASSIGN INPUTS.PresSelCalStbd[9]:=(FALSE); editable
rectangle at (125,245)-(196,266): text "1: %.0f %%"; shows PARAMS.stW1210Cfg.Spd1[1]; runs INTERN ASSIGN INPUTS.PresSelCalStbd[9]:=(FALSE); editable
rectangle at (125,230)-(196,246): text "V3 Spd - %s"; shows MAIN.fbW1210.Spd1
rectangle at (125,300)-(196,321): text "1: %.0f %%"; shows PARAMS.stW1210Cfg.Spd2[1]; runs INTERN ASSIGN INPUTS.PresSelCalStbd[9]:=(FALSE); editable
rectangle at (125,320)-(196,341): text "7: %.0f %%"; shows PARAMS.stW1210Cfg.Spd2[7]; runs INTERN ASSIGN INPUTS.PresSelCalStbd[9]:=(FALSE); editable
rounded rectangle at (130,415)-(191,446): text "SPEED / A/B"; toggles PARAMS.stW1210Cfg.A_Spd1
rectangle at (125,285)-(196,301): text "V2 Spd - %s"; shows MAIN.fbW1210.Spd2
rectangle at (125,265)-(196,286): text "7: %.0f %%"; shows PARAMS.stW1210Cfg.Spd1[7]; runs INTERN ASSIGN INPUTS.PresSelCalStbd[9]:=(FALSE); editable
rectangle at (705,135)-(776,156): text "%.0f bar"; shows PARAMS.stW1202Cfg.P1_Max; runs INTERN ASSIGN INPUTS.PresSelCalStbd[9]:=(FALSE); editable
rectangle at (515,135)-(586,156): text "%.0f bar"; shows PARAMS.stW1204Cfg.P1_Max; runs INTERN ASSIGN INPUTS.PresSelCalStbd[9]:=(FALSE); editable
rectangle at (415,135)-(486,156): text "%.0f bar"; shows PARAMS.stW1206Cfg.P1_Max; runs INTERN ASSIGN INPUTS.PresSelCalStbd[9]:=(FALSE); editable
rectangle at (30,135)-(101,156): text "%.0f bar"; shows PARAMS.stW1208Cfg.P1_Max; runs INTERN ASSIGN INPUTS.PresSelCalStbd[9]:=(FALSE); editable
rectangle at (30,120)-(101,136): text "V3 Press Max"
rectangle at (30,155)-(101,171): text "V2 Press Max"
rectangle at (125,135)-(196,156): text "%.0f bar"; shows PARAMS.stW1210Cfg.P1_Max; runs INTERN ASSIGN INPUTS.PresSelCalStbd[9]:=(FALSE); editable
rectangle at (220,135)-(291,156): text "%.0f bar"; shows PARAMS.stW1212Cfg.P1_Max; runs INTERN ASSIGN INPUTS.PresSelCalStbd[9]:=(FALSE); editable
rectangle at (315,135)-(386,156): text "%.0f bar"; shows PARAMS.stW1214Cfg.P1_Max; runs INTERN ASSIGN INPUTS.PresSelCalStbd[9]:=(FALSE); editable
rectangle at (800,135)-(871,156): text "%.0f bar"; shows PARAMS.stW1602Cfg.P1_Max; runs INTERN ASSIGN INPUTS.PresSelCalStbd[9]:=(FALSE); editable
rectangle at (610,135)-(681,156): text "%.0f bar"; shows PARAMS.stW1604Cfg.P1_Max; runs INTERN ASSIGN INPUTS.PresSelCalStbd[9]:=(FALSE); editable
rectangle at (520,55)-(581,81): text "PIT / STBD"
rectangle at (420,60)-(481,81): text "MAIN"
rectangle at (35,55)-(96,81): text "RUNNER / PORT"
rectangle at (320,55)-(381,81): text "PIT / PORT"
rectangle at (805,55)-(866,81): text "RUNNER / STBD"
rectangle at (610,55)-(681,81): text "SECONDARY / STBD"
rectangle at (220,55)-(291,81): text "SECONDARY / PORT"
rectangle at (710,55)-(771,81): text "PRIMARY / STBD"
rectangle at (130,55)-(191,81): text "PRIMARY / PORT"
rectangle at (125,80)-(196,96): text "Time Max"
rectangle at (125,120)-(196,136): text "V3 Press Max"
rectangle at (125,155)-(196,171): text "V2 Press Max"
rectangle at (220,80)-(291,96): text "Time Max"
rectangle at (220,120)-(291,136): text "V3 Press Max"
rectangle at (220,155)-(291,171): text "V2 Press Max"
rectangle at (315,80)-(386,96): text "Time Max"
rectangle at (315,120)-(386,136): text "V3 Press Max"
rectangle at (315,155)-(386,171): text "V2 Press Max"
rectangle at (415,80)-(486,96): text "Time Max"
rectangle at (415,120)-(486,136): text "V3 Press Max"
rectangle at (415,155)-(486,171): text "V2 Press Max"
rectangle at (515,80)-(586,96): text "Time Max"
rectangle at (515,120)-(586,136): text "V3 Press Max"
rectangle at (515,155)-(586,171): text "V2 Press Max"
rectangle at (610,80)-(681,96): text "Time Max"
rectangle at (610,120)-(681,136): text "V3 Press Max"
rectangle at (610,155)-(681,171): text "V2 Press Max"
rectangle at (705,80)-(776,96): text "Time Max"
rectangle at (705,120)-(776,136): text "V3 Press Max"
rectangle at (705,155)-(776,171): text "V2 Press Max"
rectangle at (800,80)-(871,96): text "Time Max"
rectangle at (800,120)-(871,136): text "V3 Press Max"
rectangle at (800,155)-(871,171): text "V2 Press Max"
rectangle at (30,475)-(101,491): text "%.1f h"; shows MAIN.W1208_UsedTime / 3600; runs INTERN ASSIGN INPUTS.PresSelCalStbd[9]:=(FALSE)
rectangle at (30,460)-(101,476): text "Used Time"
rounded rectangle at (130,500)-(191,521): text "RESET"; runs INTERN ASSIGN MAIN.W1210_UsedTime:=(0)
rectangle at (125,475)-(196,491): text "%.1f h"; shows MAIN.W1210_UsedTime / 3600; runs INTERN ASSIGN INPUTS.PresSelCalStbd[9]:=(FALSE)
rectangle at (125,460)-(196,476): text "Used Time"
rounded rectangle at (225,500)-(286,521): text "RESET"; runs INTERN ASSIGN MAIN.W1212_UsedTime:=(0)
rectangle at (220,475)-(291,491): text "%.1f h"; shows MAIN.W1212_UsedTime / 3600; runs INTERN ASSIGN INPUTS.PresSelCalStbd[9]:=(FALSE)
rectangle at (220,460)-(291,476): text "Used Time"
rounded rectangle at (320,500)-(381,521): text "RESET"; runs INTERN ASSIGN MAIN.W1214_UsedTime:=(0)
rectangle at (315,475)-(386,491): text "%.1f h"; shows MAIN.W1214_UsedTime / 3600; runs INTERN ASSIGN INPUTS.PresSelCalStbd[9]:=(FALSE)
rectangle at (315,460)-(386,476): text "Used Time"
rounded rectangle at (420,500)-(481,521): text "RESET"; runs INTERN ASSIGN MAIN.W1206_UsedTime:=(0)
rectangle at (415,475)-(486,491): text "%.1f h"; shows MAIN.W1206_UsedTime / 3600; runs INTERN ASSIGN INPUTS.PresSelCalStbd[9]:=(FALSE)
rectangle at (415,460)-(486,476): text "Used Time"
rounded rectangle at (520,500)-(581,521): text "RESET"; runs INTERN ASSIGN MAIN.W1204_UsedTime:=(0)
rectangle at (515,475)-(586,491): text "%.1f h"; shows MAIN.W1204_UsedTime / 3600; runs INTERN ASSIGN INPUTS.PresSelCalStbd[9]:=(FALSE)
rectangle at (515,460)-(586,476): text "Used Time"
rounded rectangle at (615,500)-(676,521): text "RESET"; runs INTERN ASSIGN MAIN.W1604_UsedTime:=(0)
rectangle at (610,475)-(681,491): text "%.1f h"; shows MAIN.W1604_UsedTime / 3600; runs INTERN ASSIGN INPUTS.PresSelCalStbd[9]:=(FALSE)
rectangle at (610,460)-(681,476): text "Used Time"
rounded rectangle at (710,500)-(771,521): text "RESET"; runs INTERN ASSIGN MAIN.W1202_UsedTime:=(0)
rectangle at (705,475)-(776,491): text "%.1f h"; shows MAIN.W1202_UsedTime / 3600; runs INTERN ASSIGN INPUTS.PresSelCalStbd[9]:=(FALSE)
rectangle at (705,460)-(776,476): text "Used Time"
rounded rectangle at (805,500)-(866,521): text "RESET"; runs INTERN ASSIGN MAIN.W1602_UsedTime:=(0)
rectangle at (800,475)-(871,491): text "%.1f h"; shows MAIN.W1602_UsedTime / 3600; runs INTERN ASSIGN INPUTS.PresSelCalStbd[9]:=(FALSE)
rectangle at (800,460)-(871,476): text "Used Time"
rectangle at (705,170)-(776,191): text "%.0f bar"; shows PARAMS.stW1202Cfg.P2_Max; runs INTERN ASSIGN INPUTS.PresSelCalStbd[9]:=(FALSE); editable
rectangle at (515,170)-(586,191): text "%.0f bar"; shows PARAMS.stW1204Cfg.P2_Max; runs INTERN ASSIGN INPUTS.PresSelCalStbd[9]:=(FALSE); editable
rectangle at (415,170)-(486,191): text "%.0f bar"; shows PARAMS.stW1206Cfg.P2_Max; runs INTERN ASSIGN INPUTS.PresSelCalStbd[9]:=(FALSE); editable
rectangle at (30,170)-(101,191): text "%.0f bar"; shows PARAMS.stW1208Cfg.P2_Max; runs INTERN ASSIGN INPUTS.PresSelCalStbd[9]:=(FALSE); editable
rectangle at (125,170)-(196,191): text "%.0f bar"; shows PARAMS.stW1210Cfg.P2_Max; runs INTERN ASSIGN INPUTS.PresSelCalStbd[9]:=(FALSE); editable
rectangle at (220,170)-(291,191): text "%.0f bar"; shows PARAMS.stW1212Cfg.P2_Max; runs INTERN ASSIGN INPUTS.PresSelCalStbd[9]:=(FALSE); editable
rectangle at (315,170)-(386,191): text "%.0f bar"; shows PARAMS.stW1214Cfg.P2_Max; runs INTERN ASSIGN INPUTS.PresSelCalStbd[9]:=(FALSE); editable
rectangle at (800,170)-(871,191): text "%.0f bar"; shows PARAMS.stW1602Cfg.P2_Max; runs INTERN ASSIGN INPUTS.PresSelCalStbd[9]:=(FALSE); editable
rectangle at (610,170)-(681,191): text "%.0f bar"; shows PARAMS.stW1604Cfg.P2_Max; runs INTERN ASSIGN INPUTS.PresSelCalStbd[9]:=(FALSE); editable
rectangle at (705,205)-(776,226): text "%.0f bar"; shows PARAMS.stW1202Cfg.P3_Max; runs INTERN ASSIGN INPUTS.PresSelCalStbd[9]:=(FALSE); editable
rectangle at (415,205)-(486,226): text "%.0f bar"; shows PARAMS.stW1206Cfg.P3_Max; runs INTERN ASSIGN INPUTS.PresSelCalStbd[9]:=(FALSE); editable
rectangle at (30,205)-(101,226): text "%.0f bar"; shows PARAMS.stW1208Cfg.P3_Max; runs INTERN ASSIGN INPUTS.PresSelCalStbd[9]:=(FALSE); editable
rectangle at (30,190)-(101,206): text "V1 Press Max"
rectangle at (125,205)-(196,226): text "%.0f bar"; shows PARAMS.stW1210Cfg.P3_Max; runs INTERN ASSIGN INPUTS.PresSelCalStbd[9]:=(FALSE); editable
rectangle at (220,205)-(291,226): text "%.0f bar"; shows PARAMS.stW1212Cfg.P3_Max; runs INTERN ASSIGN INPUTS.PresSelCalStbd[9]:=(FALSE); editable
rectangle at (800,205)-(871,226): text "%.0f bar"; shows PARAMS.stW1602Cfg.P3_Max; runs INTERN ASSIGN INPUTS.PresSelCalStbd[9]:=(FALSE); editable
rectangle at (610,205)-(681,226): text "%.0f bar"; shows PARAMS.stW1604Cfg.P3_Max; runs INTERN ASSIGN INPUTS.PresSelCalStbd[9]:=(FALSE); editable
rectangle at (125,190)-(196,206): text "V1 Press Max"
rectangle at (220,190)-(291,206): text "V1 Press Max"
rectangle at (415,190)-(486,206): text "V1 Press Max"
rectangle at (610,190)-(681,206): text "V1 Press Max"
rectangle at (705,190)-(776,206): text "V1 Press Max"
rectangle at (800,190)-(871,206): text "V1 Press Max"
rounded rectangle at (35,500)-(96,521): text "RESET"; runs INTERN ASSIGN MAIN.W1208_UsedTime:=(0)
rectangle at (705,355)-(776,376): text "1: %.0f %%"; shows PARAMS.stW1202Cfg.Spd3[1]; runs INTERN ASSIGN INPUTS.PresSelCalStbd[9]:=(FALSE); editable
rectangle at (705,375)-(776,396): text "7: %.0f %%"; shows PARAMS.stW1202Cfg.Spd3[7]; runs INTERN ASSIGN INPUTS.PresSelCalStbd[9]:=(FALSE); editable
rectangle at (415,355)-(486,376): text "1: %.0f %%"; shows PARAMS.stW1206Cfg.Spd3[1]; runs INTERN ASSIGN INPUTS.PresSelCalStbd[9]:=(FALSE); editable
rectangle at (415,375)-(486,396): text "7: %.0f %%"; shows PARAMS.stW1206Cfg.Spd3[7]; runs INTERN ASSIGN INPUTS.PresSelCalStbd[9]:=(FALSE); editable
rectangle at (30,355)-(101,376): text "1: %.0f %%"; shows PARAMS.stW1208Cfg.Spd3[1]; runs INTERN ASSIGN INPUTS.PresSelCalStbd[9]:=(FALSE); editable
rectangle at (30,375)-(101,396): text "7: %.0f %%"; shows PARAMS.stW1208Cfg.Spd3[7]; runs INTERN ASSIGN INPUTS.PresSelCalStbd[9]:=(FALSE); editable
rectangle at (800,355)-(871,376): text "1: %.0f %%"; shows PARAMS.stW1602Cfg.Spd3[1]; runs INTERN ASSIGN INPUTS.PresSelCalStbd[9]:=(FALSE); editable
rectangle at (800,375)-(871,396): text "7: %.0f %%"; shows PARAMS.stW1602Cfg.Spd3[7]; runs INTERN ASSIGN INPUTS.PresSelCalStbd[9]:=(FALSE); editable
rectangle at (610,355)-(681,376): text "1: %.0f %%"; shows PARAMS.stW1604Cfg.Spd3[1]; runs INTERN ASSIGN INPUTS.PresSelCalStbd[9]:=(FALSE); editable
rectangle at (610,375)-(681,396): text "7: %.0f %%"; shows PARAMS.stW1604Cfg.Spd3[7]; runs INTERN ASSIGN INPUTS.PresSelCalStbd[9]:=(FALSE); editable
rectangle at (220,355)-(291,376): text "1: %.0f %%"; shows PARAMS.stW1212Cfg.Spd3[1]; runs INTERN ASSIGN INPUTS.PresSelCalStbd[9]:=(FALSE); editable
rectangle at (220,375)-(291,396): text "7: %.0f %%"; shows PARAMS.stW1212Cfg.Spd3[7]; runs INTERN ASSIGN INPUTS.PresSelCalStbd[9]:=(FALSE); editable
rectangle at (125,355)-(196,376): text "1: %.0f %%"; shows PARAMS.stW1210Cfg.Spd3[1]; runs INTERN ASSIGN INPUTS.PresSelCalStbd[9]:=(FALSE); editable
rectangle at (125,375)-(196,396): text "7: %.0f %%"; shows PARAMS.stW1210Cfg.Spd3[7]; runs INTERN ASSIGN INPUTS.PresSelCalStbd[9]:=(FALSE); editable
rectangle at (705,340)-(776,356): text "V1 Spd - %s"; shows MAIN.fbW1202.Spd1
rectangle at (415,340)-(486,356): text "V1 Spd - %s"; shows MAIN.fbW1206.Spd1
rectangle at (30,340)-(101,356): text "V1 Spd - %s"; shows MAIN.fbW1208.Spd1
rectangle at (800,340)-(871,356): text "V1 Spd - %s"; shows MAIN.fbW1602.Spd1
rectangle at (610,340)-(681,356): text "V1 Spd - %s"; shows MAIN.fbW1604.Spd1
rectangle at (220,340)-(291,356): text "V1 Spd - %s"; shows MAIN.fbW1212.Spd1
rectangle at (125,340)-(196,356): text "V1 Spd - %s"; shows MAIN.fbW1210.Spd1
14 more shapes without text or variables
*)

(* Visualisation VISU_MAST_SETUP
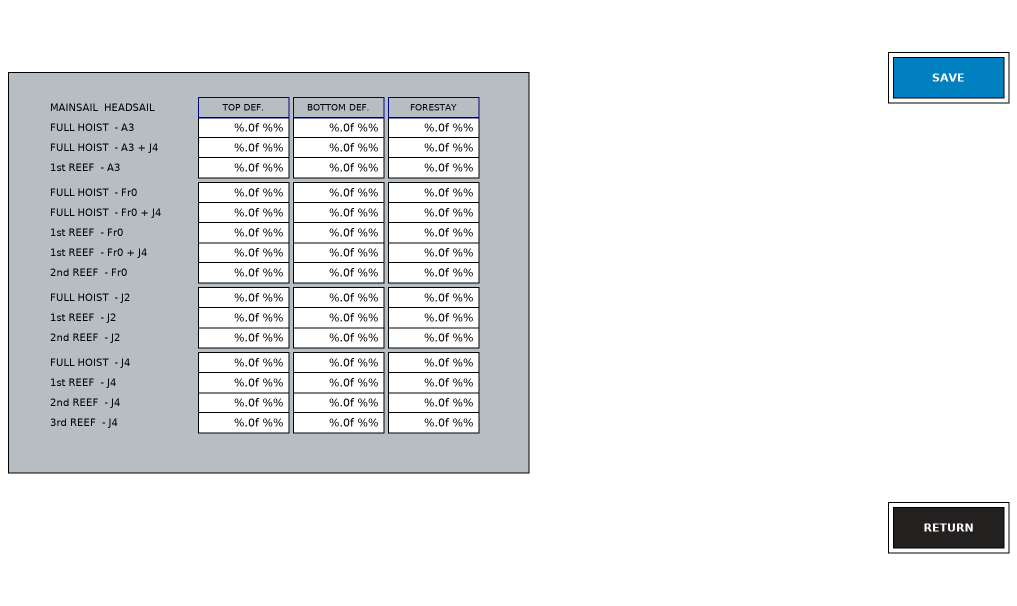
rectangle at (20,0)-(331,51): text "MAST SETUP"
rectangle at (20,550)-(331,601): text "%s"; shows INPUTS.sVisuTime
rounded rectangle at (905,55)-(1016,96): text "SAVE"; alarm colour if PARAMS.Save; toggles PARAMS.Save
rounded rectangle at (905,505)-(1016,546): text "RETURN"; opens VISU_1_CYLINDERS1
rectangle at (210,115)-(301,136): text "%.0f %%"; shows PARAMS.stMastSetup.aTDef[4,1]; runs INTERN ASSIGN INPUTS.PresSelCalStbd[9]:=(FALSE); editable
rectangle at (210,135)-(301,156): text "%.0f %%"; shows PARAMS.stMastSetup.aTDef[4,5]; runs INTERN ASSIGN INPUTS.PresSelCalStbd[9]:=(FALSE); editable
rectangle at (210,180)-(301,201): text "%.0f %%"; shows PARAMS.stMastSetup.aTDef[4,2]; runs INTERN ASSIGN INPUTS.PresSelCalStbd[9]:=(FALSE); editable
rectangle at (210,200)-(301,221): text "%.0f %%"; shows PARAMS.stMastSetup.aTDef[4,6]; runs INTERN ASSIGN INPUTS.PresSelCalStbd[9]:=(FALSE); editable
rectangle at (60,115)-(191,136): text "FULL HOIST	- A3"; shows RECV_J1939.F004.DriverDemandTorque
rectangle at (60,180)-(191,201): text "FULL HOIST	- Fr0"; shows RECV_J1939.F004.DriverDemandTorque
rectangle at (60,200)-(191,221): text "FULL HOIST	- Fr0 + J4"; shows RECV_J1939.F004.DriverDemandTorque
rectangle at (210,240)-(301,261): text "%.0f %%"; shows PARAMS.stMastSetup.aTDef[1,6]; runs INTERN ASSIGN INPUTS.PresSelCalStbd[9]:=(FALSE); editable
rectangle at (210,260)-(301,281): text "%.0f %%"; shows PARAMS.stMastSetup.aTDef[2,2]; runs INTERN ASSIGN INPUTS.PresSelCalStbd[9]:=(FALSE); editable
rectangle at (60,240)-(191,261): text "1st REEF	- Fr0 + J4"; shows RECV_J1939.F004.DriverDemandTorque
rectangle at (60,260)-(191,281): text "2nd REEF	- Fr0"; shows RECV_J1939.F004.DriverDemandTorque
rectangle at (210,155)-(301,176): text "%.0f %%"; shows PARAMS.stMastSetup.aTDef[1,1]; runs INTERN ASSIGN INPUTS.PresSelCalStbd[9]:=(FALSE); editable
rectangle at (60,155)-(191,176): text "1st REEF	- A3"; shows RECV_J1939.F004.DriverDemandTorque
rectangle at (730,550)-(896,601): text "SAVED!"; invisible if PARAMS.Saved
rectangle at (210,220)-(301,241): text "%.0f %%"; shows PARAMS.stMastSetup.aTDef[1,2]; runs INTERN ASSIGN INPUTS.PresSelCalStbd[9]:=(FALSE); editable
rectangle at (60,220)-(191,241): text "1st REEF	- Fr0"; shows RECV_J1939.F004.DriverDemandTorque
rectangle at (60,135)-(191,156): text "FULL HOIST	- A3 + J4"; shows RECV_J1939.F004.DriverDemandTorque
rectangle at (210,95)-(301,116): text "TOP DEF."
rectangle at (210,285)-(301,306): text "%.0f %%"; shows PARAMS.stMastSetup.aTDef[4,3]; runs INTERN ASSIGN INPUTS.PresSelCalStbd[9]:=(FALSE); editable
rectangle at (210,325)-(301,346): text "%.0f %%"; shows PARAMS.stMastSetup.aTDef[2,3]; runs INTERN ASSIGN INPUTS.PresSelCalStbd[9]:=(FALSE); editable
rectangle at (210,305)-(301,326): text "%.0f %%"; shows PARAMS.stMastSetup.aTDef[1,3]; runs INTERN ASSIGN INPUTS.PresSelCalStbd[9]:=(FALSE); editable
rectangle at (60,285)-(191,306): text "FULL HOIST	- J2"; shows RECV_J1939.F004.DriverDemandTorque
rectangle at (60,305)-(191,326): text "1st REEF	- J2"; shows RECV_J1939.F004.DriverDemandTorque
rectangle at (60,325)-(191,346): text "2nd REEF	- J2"; shows RECV_J1939.F004.DriverDemandTorque
rectangle at (210,350)-(301,371): text "%.0f %%"; shows PARAMS.stMastSetup.aTDef[4,4]; runs INTERN ASSIGN INPUTS.PresSelCalStbd[9]:=(FALSE); editable
rectangle at (210,390)-(301,411): text "%.0f %%"; shows PARAMS.stMastSetup.aTDef[2,4]; runs INTERN ASSIGN INPUTS.PresSelCalStbd[9]:=(FALSE); editable
rectangle at (210,370)-(301,391): text "%.0f %%"; shows PARAMS.stMastSetup.aTDef[1,4]; runs INTERN ASSIGN INPUTS.PresSelCalStbd[9]:=(FALSE); editable
rectangle at (60,350)-(191,371): text "FULL HOIST	- J4"; shows RECV_J1939.F004.DriverDemandTorque
rectangle at (60,370)-(191,391): text "1st REEF	- J4"; shows RECV_J1939.F004.DriverDemandTorque
rectangle at (60,390)-(191,411): text "2nd REEF	- J4"; shows RECV_J1939.F004.DriverDemandTorque
rectangle at (210,410)-(301,431): text "%.0f %%"; shows PARAMS.stMastSetup.aTDef[3,4]; runs INTERN ASSIGN INPUTS.PresSelCalStbd[9]:=(FALSE); editable
rectangle at (60,410)-(191,431): text "3rd REEF	- J4"; shows RECV_J1939.F004.DriverDemandTorque
rectangle at (60,95)-(206,116): text "MAINSAIL	HEADSAIL"; shows RECV_J1939.F004.DriverDemandTorque
rectangle at (305,115)-(396,136): text "%.0f %%"; shows PARAMS.stMastSetup.aBDef[4,1]; runs INTERN ASSIGN INPUTS.PresSelCalStbd[9]:=(FALSE); editable
rectangle at (305,135)-(396,156): text "%.0f %%"; shows PARAMS.stMastSetup.aBDef[4,5]; runs INTERN ASSIGN INPUTS.PresSelCalStbd[9]:=(FALSE); editable
rectangle at (305,180)-(396,201): text "%.0f %%"; shows PARAMS.stMastSetup.aBDef[4,2]; runs INTERN ASSIGN INPUTS.PresSelCalStbd[9]:=(FALSE); editable
rectangle at (305,200)-(396,221): text "%.0f %%"; shows PARAMS.stMastSetup.aBDef[4,6]; runs INTERN ASSIGN INPUTS.PresSelCalStbd[9]:=(FALSE); editable
rectangle at (305,240)-(396,261): text "%.0f %%"; shows PARAMS.stMastSetup.aBDef[1,6]; runs INTERN ASSIGN INPUTS.PresSelCalStbd[9]:=(FALSE); editable
rectangle at (305,260)-(396,281): text "%.0f %%"; shows PARAMS.stMastSetup.aBDef[2,2]; runs INTERN ASSIGN INPUTS.PresSelCalStbd[9]:=(FALSE); editable
rectangle at (305,155)-(396,176): text "%.0f %%"; shows PARAMS.stMastSetup.aBDef[1,1]; runs INTERN ASSIGN INPUTS.PresSelCalStbd[9]:=(FALSE); editable
rectangle at (305,220)-(396,241): text "%.0f %%"; shows PARAMS.stMastSetup.aBDef[1,2]; runs INTERN ASSIGN INPUTS.PresSelCalStbd[9]:=(FALSE); editable
rectangle at (305,95)-(396,116): text "BOTTOM DEF."
rectangle at (305,285)-(396,306): text "%.0f %%"; shows PARAMS.stMastSetup.aBDef[4,3]; runs INTERN ASSIGN INPUTS.PresSelCalStbd[9]:=(FALSE); editable
rectangle at (305,325)-(396,346): text "%.0f %%"; shows PARAMS.stMastSetup.aBDef[2,3]; runs INTERN ASSIGN INPUTS.PresSelCalStbd[9]:=(FALSE); editable
rectangle at (305,305)-(396,326): text "%.0f %%"; shows PARAMS.stMastSetup.aBDef[1,3]; runs INTERN ASSIGN INPUTS.PresSelCalStbd[9]:=(FALSE); editable
rectangle at (305,350)-(396,371): text "%.0f %%"; shows PARAMS.stMastSetup.aBDef[4,4]; runs INTERN ASSIGN INPUTS.PresSelCalStbd[9]:=(FALSE); editable
rectangle at (305,390)-(396,411): text "%.0f %%"; shows PARAMS.stMastSetup.aBDef[2,4]; runs INTERN ASSIGN INPUTS.PresSelCalStbd[9]:=(FALSE); editable
rectangle at (305,370)-(396,391): text "%.0f %%"; shows PARAMS.stMastSetup.aBDef[1,4]; runs INTERN ASSIGN INPUTS.PresSelCalStbd[9]:=(FALSE); editable
rectangle at (305,410)-(396,431): text "%.0f %%"; shows PARAMS.stMastSetup.aBDef[3,4]; runs INTERN ASSIGN INPUTS.PresSelCalStbd[9]:=(FALSE); editable
rectangle at (400,115)-(491,136): text "%.0f %%"; shows PARAMS.stMastSetup.aFSY[4,1]; runs INTERN ASSIGN INPUTS.PresSelCalStbd[9]:=(FALSE); editable
rectangle at (400,135)-(491,156): text "%.0f %%"; shows PARAMS.stMastSetup.aFSY[4,5]; runs INTERN ASSIGN INPUTS.PresSelCalStbd[9]:=(FALSE); editable
rectangle at (400,180)-(491,201): text "%.0f %%"; shows PARAMS.stMastSetup.aFSY[4,2]; runs INTERN ASSIGN INPUTS.PresSelCalStbd[9]:=(FALSE); editable
rectangle at (400,200)-(491,221): text "%.0f %%"; shows PARAMS.stMastSetup.aFSY[4,6]; runs INTERN ASSIGN INPUTS.PresSelCalStbd[9]:=(FALSE); editable
rectangle at (400,240)-(491,261): text "%.0f %%"; shows PARAMS.stMastSetup.aFSY[1,6]; runs INTERN ASSIGN INPUTS.PresSelCalStbd[9]:=(FALSE); editable
rectangle at (400,260)-(491,281): text "%.0f %%"; shows PARAMS.stMastSetup.aFSY[2,2]; runs INTERN ASSIGN INPUTS.PresSelCalStbd[9]:=(FALSE); editable
rectangle at (400,155)-(491,176): text "%.0f %%"; shows PARAMS.stMastSetup.aFSY[1,1]; runs INTERN ASSIGN INPUTS.PresSelCalStbd[9]:=(FALSE); editable
rectangle at (400,220)-(491,241): text "%.0f %%"; shows PARAMS.stMastSetup.aFSY[1,2]; runs INTERN ASSIGN INPUTS.PresSelCalStbd[9]:=(FALSE); editable
rectangle at (400,95)-(491,116): text "FORESTAY"
rectangle at (400,285)-(491,306): text "%.0f %%"; shows PARAMS.stMastSetup.aFSY[4,3]; runs INTERN ASSIGN INPUTS.PresSelCalStbd[9]:=(FALSE); editable
rectangle at (400,325)-(491,346): text "%.0f %%"; shows PARAMS.stMastSetup.aFSY[2,3]; runs INTERN ASSIGN INPUTS.PresSelCalStbd[9]:=(FALSE); editable
rectangle at (400,305)-(491,326): text "%.0f %%"; shows PARAMS.stMastSetup.aFSY[1,3]; runs INTERN ASSIGN INPUTS.PresSelCalStbd[9]:=(FALSE); editable
rectangle at (400,350)-(491,371): text "%.0f %%"; shows PARAMS.stMastSetup.aFSY[4,4]; runs INTERN ASSIGN INPUTS.PresSelCalStbd[9]:=(FALSE); editable
rectangle at (400,390)-(491,411): text "%.0f %%"; shows PARAMS.stMastSetup.aFSY[2,4]; runs INTERN ASSIGN INPUTS.PresSelCalStbd[9]:=(FALSE); editable
rectangle at (400,370)-(491,391): text "%.0f %%"; shows PARAMS.stMastSetup.aFSY[1,4]; runs INTERN ASSIGN INPUTS.PresSelCalStbd[9]:=(FALSE); editable
rectangle at (400,410)-(491,431): text "%.0f %%"; shows PARAMS.stMastSetup.aFSY[3,4]; runs INTERN ASSIGN INPUTS.PresSelCalStbd[9]:=(FALSE); editable
3 more shapes without text or variables
*)
